LIN {X 0,Y 128.631,Z 703.14,A -85,B 0,C 180,E1 -30051.999,E2 -30051.999} C_VEL
LIN {X 0,Y 134.628,Z 692.341,A -85,B 0,C 180,E1 -30052.672,E2 -30052.672} C_VEL
LIN {X 0,Y 139.361,Z 682.091,A -85,B 0,C 180,E1 -30053.131,E2 -30053.131} C_VEL
LIN {X 0,Y 143.551,Z 670.824,A -85,B 0,C 180,E1 -30053.508,E2 -30053.508} C_VEL
LIN {X 0,Y 146.834,Z 659.297,A -85,B 0,C 180,E1 -30053.808,E2 -30053.808} C_VEL
LIN {X 0,Y 148.842,Z 649.788,A -85,B 0,C 180,E1 -30054.037,E2 -30054.037} C_VEL
LIN {X 0,Y 148.62,Z 648.347,A -85,B 0,C 180,E1 -30055.938,E2 -30055.938} C_VEL
LIN {X 0,Y 148.514,Z 646.401,A -85,B 0,C 180,E1 -30059.999,E2 -30059.999} C_VEL
LIN {X 0,Y 148.714,Z 649.137,A -85,B 0,C 180,E1 -30065.592,E2 -30065.592} C_VEL
LIN {X 0,Y 149.267,Z 652.354,A -85,B 0,C 180,E1 -30069.107,E2 -30069.107} C_VEL
LIN {X 0,Y 149.738,Z 657.139,A -85,B 0,C 180,E1 -30072.527,E2 -30072.527} C_VEL
LIN {X 0,Y 150.095,Z 661.69,A -85,B 0,C 180,E1 -30074.922,E2 -30074.922} C_VEL
LIN {X 0,Y 149.921,Z 667.758,A -85,B 0,C 180,E1 -30077.387,E2 -30077.387} C_VEL
LIN {X 0,Y 149.394,Z 677.527,A -85,B 0,C 180,E1 -30081.047,E2 -30081.047} C_VEL
LIN {X 0,Y 149.068,Z 687.198,A -85,B 0,C 180,E1 -30085.106,E2 -30085.106} C_VEL
LIN {X 0,Y 149.259,Z 696.603,A -85,B 0,C 180,E1 -30089.604,E2 -30089.604} C_VEL
LIN {X 0,Y 150.212,Z 704.997,A -85,B 0,C 180,E1 -30094.154,E2 -30094.154} C_VEL
LIN {X 0,Y 152.27,Z 713.653,A -85,B 0,C 180,E1 -30099.39,E2 -30099.39} C_VEL
LIN {X 0,Y 155.461,Z 721.258,A -85,B 0,C 180,E1 -30104.481,E2 -30104.481} C_VEL
LIN {X 0,Y 160.455,Z 728.846,A -85,B 0,C 180,E1 -30110.039,E2 -30110.039} C_VEL
LIN {X 0,Y 167.763,Z 736.335,A -85,B 0,C 180,E1 -30115.979,E2 -30115.979} C_VEL
LIN {X 0,Y 169.712,Z 738.673,A -85,B 0,C 180,E1 -30117.709,E2 -30117.709} C_VEL
LIN {X 0,Y 173.531,Z 746.392,A -85,B 0,C 180,E1 -30122.934,E2 -30122.934} C_VEL
LIN {X 0,Y 176.298,Z 748.654,A -85,B 0,C 180,E1 -30124.847,E2 -30124.847} C_VEL
LIN {X 0,Y 176.824,Z 748.877,A -85,B 0,C 180,E1 -30125.101,E2 -30125.101} C_VEL
LIN {X 0,Y 192.712,Z 754.942,A -85,B 0,C 180,E1 -30131.472,E2 -30131.472} C_VEL
LIN {X 0,Y 203.581,Z 758.254,A -85,B 0,C 180,E1 -30135.149,E2 -30135.149} C_VEL
LIN {X 0,Y 209.199,Z 759.811,A -85,B 0,C 180,E1 -30136.965,E2 -30136.965} C_VEL
LIN {X 0,Y 214.899,Z 761.328,A -85,B 0,C 180,E1 -30138.841,E2 -30138.841} C_VEL
LIN {X 0,Y 220.679,Z 762.865,A -85,B 0,C 180,E1 -30140.838,E2 -30140.838} C_VEL
LIN {X 0,Y 226.507,Z 764.368,A -85,B 0,C 180,E1 -30143.153,E2 -30143.153} C_VEL
LIN {X 0,Y 229.657,Z 765.23,A -85,B 0,C 180,E1 -30144.733,E2 -30144.733} C_VEL
LIN {X 0,Y 232.744,Z 765.966,A -85,B 0,C 180,E1 -30146.538,E2 -30146.538} C_VEL
LIN {X 0,Y 234.8,Z 766.382,A -85,B 0,C 180,E1 -30148.285,E2 -30148.285} C_VEL
LIN {X 0,Y 236.127,Z 766.522,A -85,B 0,C 180,E1 -30150,E2 -30150} C_VEL
LIN {X 0,Y 234.811,Z 766.381,A -85,B 0,C 180,E1 -30151.715,E2 -30151.715} C_VEL
LIN {X 0,Y 232.396,Z 765.889,A -85,B 0,C 180,E1 -30153.669,E2 -30153.669} C_VEL
LIN {X 0,Y 229.683,Z 765.23,A -85,B 0,C 180,E1 -30155.267,E2 -30155.267} C_VEL
LIN {X 0,Y 225.823,Z 764.189,A -85,B 0,C 180,E1 -30157.151,E2 -30157.151} C_VEL
LIN {X 0,Y 220.686,Z 762.857,A -85,B 0,C 180,E1 -30159.173,E2 -30159.173} C_VEL
LIN {X 0,Y 214.372,Z 761.188,A -85,B 0,C 180,E1 -30161.344,E2 -30161.344} C_VEL
LIN {X 0,Y 207.029,Z 759.205,A -85,B 0,C 180,E1 -30163.746,E2 -30163.746} C_VEL
LIN {X 0,Y 198.092,Z 756.646,A -85,B 0,C 180,E1 -30166.685,E2 -30166.685} C_VEL
LIN {X 0,Y 182.466,Z 751.292,A -85,B 0,C 180,E1 -30172.425,E2 -30172.425} C_VEL
LIN {X 0,Y 170.882,Z 745.936,A -85,B 0,C 180,E1 -30177.844,E2 -30177.844} C_VEL
LIN {X 0,Y 161.108,Z 739.323,A -85,B 0,C 180,E1 -30184.023,E2 -30184.023} C_VEL
LIN {X 0,Y 154.807,Z 733.026,A -85,B 0,C 180,E1 -30189.489,E2 -30189.489} C_VEL
LIN {X 0,Y 149.927,Z 725.802,A -85,B 0,C 180,E1 -30195.322,E2 -30195.322} C_VEL
LIN {X 0,Y 146.606,Z 717.429,A -85,B 0,C 180,E1 -30201.452,E2 -30201.452} C_VEL
LIN {X 0,Y 145.012,Z 708.707,A -85,B 0,C 180,E1 -30207.116,E2 -30207.116} C_VEL
LIN {X 0,Y 144.615,Z 699.602,A -85,B 0,C 180,E1 -30212.333,E2 -30212.333} C_VEL
LIN {X 0,Y 145.085,Z 690.28,A -85,B 0,C 180,E1 -30216.978,E2 -30216.978} C_VEL
LIN {X 0,Y 146.009,Z 680.966,A -85,B 0,C 180,E1 -30221.042,E2 -30221.042} C_VEL
LIN {X 0,Y 147.298,Z 669.426,A -85,B 0,C 180,E1 -30225.494,E2 -30225.494} C_VEL
LIN {X 0,Y 147.568,Z 663.711,A -85,B 0,C 180,E1 -30228.324,E2 -30228.324} C_VEL
LIN {X 0,Y 147.397,Z 659.445,A -85,B 0,C 180,E1 -30231.259,E2 -30231.259} C_VEL
LIN {X 0,Y 147.172,Z 656.298,A -85,B 0,C 180,E1 -30234.521,E2 -30234.521} C_VEL
LIN {X 0,Y 147.108,Z 654.875,A -85,B 0,C 180,E1 -30236.826,E2 -30236.826} C_VEL
LIN {X 0,Y 147.268,Z 653.504,A -85,B 0,C 180,E1 -30240.001,E2 -30240.001} C_VEL
LIN {X 0,Y 147.194,Z 655.069,A -85,B 0,C 180,E1 -30243.318,E2 -30243.318} C_VEL
LIN {X 0,Y 144.031,Z 667.176,A -85,B 0,C 180,E1 -30243.612,E2 -30243.612} C_VEL
LIN {X 0,Y 140,Z 678.676,A -85,B 0,C 180,E1 -30243.883,E2 -30243.883} C_VEL
LIN {X 0,Y 135.652,Z 688.64,A -85,B 0,C 180,E1 -30244.21,E2 -30244.21} C_VEL
LIN {X 0,Y 130.439,Z 698.552,A -85,B 0,C 180,E1 -30244.623,E2 -30244.623} C_VEL
LIN {X 0,Y 124.375,Z 708.269,A -85,B 0,C 180,E1 -30245.188,E2 -30245.188} C_VEL
LIN {X 0,Y 117.455,Z 717.679,A -85,B 0,C 180,E1 -30245.875,E2 -30245.875} C_VEL
LIN {X 0,Y 109.709,Z 726.693,A -85,B 0,C 180,E1 -30246.824,E2 -30246.824} C_VEL
LIN {X 0,Y 102.486,Z 734.008,A -85,B 0,C 180,E1 -30247.885,E2 -30247.885} C_VEL
LIN {X 0,Y 94.355,Z 741.184,A -85,B 0,C 180,E1 -30249.286,E2 -30249.286} C_VEL
LIN {X 0,Y 84.224,Z 748.79,A -85,B 0,C 180,E1 -30251.351,E2 -30251.351} C_VEL
LIN {X 0,Y 75.887,Z 754.19,A -85,B 0,C 180,E1 -30253.495,E2 -30253.495} C_VEL
LIN {X 0,Y 66.094,Z 759.623,A -85,B 0,C 180,E1 -30256.868,E2 -30256.868} C_VEL
LIN {X 0,Y 56.618,Z 764.075,A -85,B 0,C 180,E1 -30261.425,E2 -30261.425} C_VEL
LIN {X 0,Y 47.658,Z 767.628,A -85,B 0,C 180,E1 -30267.776,E2 -30267.776} C_VEL
LIN {X 0,Y 42.078,Z 769.575,A -85,B 0,C 180,E1 -30273.374,E2 -30273.374} C_VEL
LIN {X 0,Y 32.641,Z 772.279,A -85,B 0,C 180,E1 -30289.766,E2 -30289.766} C_VEL
LIN {X 0,Y 27.433,Z 773.598,A -85,B 0,C 180,E1 -30315.156,E2 -30315.156} C_VEL
LIN {X 0,Y 27.054,Z 773.863,A -85,B 0,C 180,E1 -30330,E2 -30330} C_VEL
LIN {X 0,Y 29.383,Z 773.111,A -85,B 0,C 180,E1 -30358.578,E2 -30358.578} C_VEL
LIN {X 0,Y 32.641,Z 772.279,A -85,B 0,C 180,E1 -30370.235,E2 -30370.235} C_VEL
LIN {X 0,Y 42.073,Z 769.575,A -85,B 0,C 180,E1 -30386.635,E2 -30386.635} C_VEL
LIN {X 0,Y 50.55,Z 766.607,A -85,B 0,C 180,E1 -30394.645,E2 -30394.645} C_VEL
LIN {X 0,Y 59.739,Z 762.774,A -85,B 0,C 180,E1 -30400.245,E2 -30400.245} C_VEL
LIN {X 0,Y 69.33,Z 758.007,A -85,B 0,C 180,E1 -30404.364,E2 -30404.364} C_VEL
LIN {X 0,Y 80.868,Z 751.063,A -85,B 0,C 180,E1 -30407.872,E2 -30407.872} C_VEL
LIN {X 0,Y 90.975,Z 743.859,A -85,B 0,C 180,E1 -30410.044,E2 -30410.044} C_VEL
LIN {X 0,Y 99.476,Z 736.792,A -85,B 0,C 180,E1 -30411.523,E2 -30411.523} C_VEL
LIN {X 0,Y 108.005,Z 728.514,A -85,B 0,C 180,E1 -30412.891,E2 -30412.891} C_VEL
LIN {X 0,Y 115.737,Z 719.798,A -85,B 0,C 180,E1 -30413.895,E2 -30413.895} C_VEL
LIN {X 0,Y 122.643,Z 710.747,A -85,B 0,C 180,E1 -30414.652,E2 -30414.652} C_VEL
LIN {X 0,Y 128.704,Z 701.478,A -85,B 0,C 180,E1 -30415.231,E2 -30415.231} C_VEL
LIN {X 0,Y 133.909,Z 692.143,A -85,B 0,C 180,E1 -30415.684,E2 -30415.684} C_VEL
LIN {X 0,Y 138.692,Z 681.893,A -85,B 0,C 180,E1 -30416.039,E2 -30416.039} C_VEL
LIN {X 0,Y 142.851,Z 670.851,A -85,B 0,C 180,E1 -30416.328,E2 -30416.328} C_VEL
LIN {X 0,Y 146.112,Z 659.636,A -85,B 0,C 180,E1 -30416.56,E2 -30416.56} C_VEL
LIN {X 0,Y 147.191,Z 655.075,A -85,B 0,C 180,E1 -30416.691,E2 -30416.691} C_VEL
LIN {X 0,Y 147.269,Z 653.498,A -85,B 0,C 180,E1 -30419.999,E2 -30419.999} C_VEL
LIN {X 0,Y 147.164,Z 655.943,A -85,B 0,C 180,E1 -30425.05,E2 -30425.05} C_VEL
LIN {X 0,Y 147.363,Z 658.957,A -85,B 0,C 180,E1 -30428.326,E2 -30428.326} C_VEL
LIN {X 0,Y 147.578,Z 662.572,A -85,B 0,C 180,E1 -30430.98,E2 -30430.98} C_VEL
LIN {X 0,Y 147.465,Z 666.324,A -85,B 0,C 180,E1 -30433.083,E2 -30433.083} C_VEL
LIN {X 0,Y 147.16,Z 671.262,A -85,B 0,C 180,E1 -30435.228,E2 -30435.228} C_VEL
LIN {X 0,Y 145.677,Z 684.666,A -85,B 0,C 180,E1 -30440.529,E2 -30440.529} C_VEL
LIN {X 0,Y 144.86,Z 694.637,A -85,B 0,C 180,E1 -30445.118,E2 -30445.118} C_VEL
LIN {X 0,Y 144.752,Z 704.962,A -85,B 0,C 180,E1 -30450.649,E2 -30450.649} C_VEL
LIN {X 0,Y 145.787,Z 713.972,A -85,B 0,C 180,E1 -30456.193,E2 -30456.193} C_VEL
LIN {X 0,Y 148.483,Z 722.834,A -85,B 0,C 180,E1 -30462.412,E2 -30462.412} C_VEL
LIN {X 0,Y 152.199,Z 729.57,A -85,B 0,C 180,E1 -30467.629,E2 -30467.629} C_VEL
LIN {X 0,Y 158.771,Z 737.265,A -85,B 0,C 180,E1 -30474.127,E2 -30474.127} C_VEL
LIN {X 0,Y 166.3,Z 743.228,A -85,B 0,C 180,E1 -30479.528,E2 -30479.528} C_VEL
LIN {X 0,Y 176.824,Z 748.877,A -85,B 0,C 180,E1 -30485.101,E2 -30485.101} C_VEL
LIN {X 0,Y 179.618,Z 750.606,A -85,B 0,C 180,E1 -30486.682,E2 -30486.682} C_VEL
LIN {X 0,Y 182.983,Z 753.911,A -85,B 0,C 180,E1 -30489.444,E2 -30489.444} C_VEL
LIN {X 0,Y 185.814,Z 756.293,A -85,B 0,C 180,E1 -30491.622,E2 -30491.622} C_VEL
LIN {X 0,Y 188.736,Z 757.733,A -85,B 0,C 180,E1 -30493.13,E2 -30493.13} C_VEL
LIN {X 0,Y 189.939,Z 758.098,A -85,B 0,C 180,E1 -30493.587,E2 -30493.587} C_VEL
LIN {X 0,Y 203.479,Z 761.495,A -85,B 0,C 180,E1 -30498.04,E2 -30498.04} C_VEL
LIN {X 0,Y 210.566,Z 763.153,A -85,B 0,C 180,E1 -30500.394,E2 -30500.394} C_VEL
LIN {X 0,Y 216.571,Z 764.444,A -85,B 0,C 180,E1 -30502.542,E2 -30502.542} C_VEL
LIN {X 0,Y 219.238,Z 764.993,A -85,B 0,C 180,E1 -30503.582,E2 -30503.582} C_VEL
LIN {X 0,Y 221.312,Z 765.463,A -85,B 0,C 180,E1 -30504.533,E2 -30504.533} C_VEL
LIN {X 0,Y 225.271,Z 766.252,A -85,B 0,C 180,E1 -30506.676,E2 -30506.676} C_VEL
LIN {X 0,Y 227.318,Z 766.587,A -85,B 0,C 180,E1 -30508.228,E2 -30508.228} C_VEL
LIN {X 0,Y 228.896,Z 766.724,A -85,B 0,C 180,E1 -30510,E2 -30510} C_VEL
LIN {X 0,Y 227.327,Z 766.587,A -85,B 0,C 180,E1 -30511.772,E2 -30511.772} C_VEL
LIN {X 0,Y 224.825,Z 766.187,A -85,B 0,C 180,E1 -30513.584,E2 -30513.584} C_VEL
LIN {X 0,Y 221.344,Z 765.462,A -85,B 0,C 180,E1 -30515.466,E2 -30515.466} C_VEL
LIN {X 0,Y 219.24,Z 764.99,A -85,B 0,C 180,E1 -30516.423,E2 -30516.423} C_VEL
LIN {X 0,Y 213.274,Z 763.724,A -85,B 0,C 180,E1 -30518.673,E2 -30518.673} C_VEL
LIN {X 0,Y 207.394,Z 762.392,A -85,B 0,C 180,E1 -30520.671,E2 -30520.671} C_VEL
LIN {X 0,Y 201.614,Z 761.075,A -85,B 0,C 180,E1 -30522.572,E2 -30522.572} C_VEL
LIN {X 0,Y 186.877,Z 757.241,A -85,B 0,C 180,E1 -30527.509,E2 -30527.509} C_VEL
LIN {X 0,Y 169.88,Z 751.256,A -85,B 0,C 180,E1 -30534.477,E2 -30534.477} C_VEL
LIN {X 0,Y 159.155,Z 745.601,A -85,B 0,C 180,E1 -30540.564,E2 -30540.564} C_VEL
LIN {X 0,Y 152.043,Z 740.176,A -85,B 0,C 180,E1 -30546.014,E2 -30546.014} C_VEL
LIN {X 0,Y 146.258,Z 733.384,A -85,B 0,C 180,E1 -30552.277,E2 -30552.277} C_VEL
LIN {X 0,Y 142.626,Z 726.672,A -85,B 0,C 180,E1 -30558.024,E2 -30558.024} C_VEL
LIN {X 0,Y 140.256,Z 717.486,A -85,B 0,C 180,E1 -30564.975,E2 -30564.975} C_VEL
LIN {X 0,Y 139.769,Z 710.287,A -85,B 0,C 180,E1 -30569.814,E2 -30569.814} C_VEL
LIN {X 0,Y 140.326,Z 700.581,A -85,B 0,C 180,E1 -30575.449,E2 -30575.449} C_VEL
LIN {X 0,Y 141.669,Z 690.542,A -85,B 0,C 180,E1 -30580.482,E2 -30580.482} C_VEL
LIN {X 0,Y 143.465,Z 680.267,A -85,B 0,C 180,E1 -30584.866,E2 -30584.866} C_VEL
LIN {X 0,Y 144.643,Z 673.944,A -85,B 0,C 180,E1 -30587.37,E2 -30587.37} C_VEL
LIN {X 0,Y 145.048,Z 669.625,A -85,B 0,C 180,E1 -30589.533,E2 -30589.533} C_VEL
LIN {X 0,Y 145.232,Z 666.495,A -85,B 0,C 180,E1 -30591.654,E2 -30591.654} C_VEL
LIN {X 0,Y 145.396,Z 663.266,A -85,B 0,C 180,E1 -30594.801,E2 -30594.801} C_VEL
LIN {X 0,Y 145.418,Z 661.848,A -85,B 0,C 180,E1 -30596.885,E2 -30596.885} C_VEL
LIN {X 0,Y 145.57,Z 660.548,A -85,B 0,C 180,E1 -30600.001,E2 -30600.001} C_VEL
LIN {X 0,Y 145.51,Z 660.875,A -85,B 0,C 180,E1 -30600.627,E2 -30600.627} C_VEL
LIN {X 0,Y 141.261,Z 674.629,A -85,B 0,C 180,E1 -30600.91,E2 -30600.91} C_VEL
LIN {X 0,Y 136.192,Z 686.69,A -85,B 0,C 180,E1 -30601.165,E2 -30601.165} C_VEL
LIN {X 0,Y 130.06,Z 698.354,A -85,B 0,C 180,E1 -30601.506,E2 -30601.506} C_VEL
LIN {X 0,Y 123.935,Z 708.071,A -85,B 0,C 180,E1 -30601.914,E2 -30601.914} C_VEL
LIN {X 0,Y 116.942,Z 717.481,A -85,B 0,C 180,E1 -30602.418,E2 -30602.418} C_VEL
LIN {X 0,Y 109.091,Z 726.494,A -85,B 0,C 180,E1 -30603.102,E2 -30603.102} C_VEL
LIN {X 0,Y 100.922,Z 734.556,A -85,B 0,C 180,E1 -30603.995,E2 -30603.995} C_VEL
LIN {X 0,Y 93.471,Z 740.986,A -85,B 0,C 180,E1 -30604.975,E2 -30604.975} C_VEL
LIN {X 0,Y 84.837,Z 747.455,A -85,B 0,C 180,E1 -30606.243,E2 -30606.243} C_VEL
LIN {X 0,Y 74.545,Z 753.99,A -85,B 0,C 180,E1 -30608.151,E2 -30608.151} C_VEL
LIN {X 0,Y 64.384,Z 759.424,A -85,B 0,C 180,E1 -30610.769,E2 -30610.769} C_VEL
LIN {X 0,Y 54.417,Z 763.874,A -85,B 0,C 180,E1 -30614.394,E2 -30614.394} C_VEL
LIN {X 0,Y 44.777,Z 767.429,A -85,B 0,C 180,E1 -30619.661,E2 -30619.661} C_VEL
LIN {X 0,Y 38.604,Z 769.376,A -85,B 0,C 180,E1 -30624.462,E2 -30624.462} C_VEL
LIN {X 0,Y 27.568,Z 772.08,A -85,B 0,C 180,E1 -30640.112,E2 -30640.112} C_VEL
LIN {X 0,Y 20.629,Z 773.399,A -85,B 0,C 180,E1 -30670.082,E2 -30670.082} C_VEL
LIN {X 0,Y 19.957,Z 773.665,A -85,B 0,C 180,E1 -30690,E2 -30690} C_VEL
LIN {X 0,Y 23.362,Z 772.912,A -85,B 0,C 180,E1 -30726.987,E2 -30726.987} C_VEL
LIN {X 0,Y 27.567,Z 772.08,A -85,B 0,C 180,E1 -30739.89,E2 -30739.89} C_VEL
LIN {X 0,Y 38.6,Z 769.375,A -85,B 0,C 180,E1 -30755.554,E2 -30755.554} C_VEL
LIN {X 0,Y 51.133,Z 765.141,A -85,B 0,C 180,E1 -30764.174,E2 -30764.174} C_VEL
LIN {X 0,Y 61.036,Z 761.004,A -85,B 0,C 180,E1 -30768.156,E2 -30768.156} C_VEL
LIN {X 0,Y 71.146,Z 755.904,A -85,B 0,C 180,E1 -30771.044,E2 -30771.044} C_VEL
LIN {X 0,Y 81.395,Z 749.728,A -85,B 0,C 180,E1 -30773.185,E2 -30773.185} C_VEL
LIN {X 0,Y 90.014,Z 743.659,A -85,B 0,C 180,E1 -30774.534,E2 -30774.534} C_VEL
LIN {X 0,Y 98.677,Z 736.593,A -85,B 0,C 180,E1 -30775.628,E2 -30775.628} C_VEL
LIN {X 0,Y 107.355,Z 728.314,A -85,B 0,C 180,E1 -30776.676,E2 -30776.676} C_VEL
LIN {X 0,Y 115.198,Z 719.6,A -85,B 0,C 180,E1 -30777.419,E2 -30777.419} C_VEL
LIN {X 0,Y 122.185,Z 710.549,A -85,B 0,C 180,E1 -30777.97,E2 -30777.97} C_VEL
LIN {X 0,Y 128.308,Z 701.28,A -85,B 0,C 180,E1 -30778.396,E2 -30778.396} C_VEL
LIN {X 0,Y 133.562,Z 691.945,A -85,B 0,C 180,E1 -30778.717,E2 -30778.717} C_VEL
LIN {X 0,Y 138.383,Z 681.695,A -85,B 0,C 180,E1 -30778.968,E2 -30778.968} C_VEL
LIN {X 0,Y 142.572,Z 670.653,A -85,B 0,C 180,E1 -30779.178,E2 -30779.178} C_VEL
LIN {X 0,Y 145.516,Z 660.849,A -85,B 0,C 180,E1 -30779.382,E2 -30779.382} C_VEL
LIN {X 0,Y 145.572,Z 660.537,A -85,B 0,C 180,E1 -30779.999,E2 -30779.999} C_VEL
LIN {X 0,Y 145.418,Z 662.581,A -85,B 0,C 180,E1 -30784.329,E2 -30784.329} C_VEL
LIN {X 0,Y 145.32,Z 664.859,A -85,B 0,C 180,E1 -30786.943,E2 -30786.943} C_VEL
LIN {X 0,Y 145.126,Z 668.458,A -85,B 0,C 180,E1 -30789.757,E2 -30789.757} C_VEL
LIN {X 0,Y 144.82,Z 672.393,A -85,B 0,C 180,E1 -30791.902,E2 -30791.902} C_VEL
LIN {X 0,Y 143.686,Z 678.991,A -85,B 0,C 180,E1 -30794.632,E2 -30794.632} C_VEL
LIN {X 0,Y 142.28,Z 687.049,A -85,B 0,C 180,E1 -30797.982,E2 -30797.982} C_VEL
LIN {X 0,Y 140.872,Z 696.007,A -85,B 0,C 180,E1 -30802.148,E2 -30802.148} C_VEL
LIN {X 0,Y 139.975,Z 704.777,A -85,B 0,C 180,E1 -30806.863,E2 -30806.863} C_VEL
LIN {X 0,Y 139.94,Z 713.697,A -85,B 0,C 180,E1 -30812.417,E2 -30812.417} C_VEL
LIN {X 0,Y 141.228,Z 722.184,A -85,B 0,C 180,E1 -30818.462,E2 -30818.462} C_VEL
LIN {X 0,Y 144.302,Z 730.211,A -85,B 0,C 180,E1 -30824.924,E2 -30824.924} C_VEL
LIN {X 0,Y 149.549,Z 737.581,A -85,B 0,C 180,E1 -30831.528,E2 -30831.528} C_VEL
LIN {X 0,Y 157.24,Z 744.344,A -85,B 0,C 180,E1 -30838.125,E2 -30838.125} C_VEL
LIN {X 0,Y 165.348,Z 749.19,A -85,B 0,C 180,E1 -30843.197,E2 -30843.197} C_VEL
LIN {X 0,Y 179.718,Z 754.967,A -85,B 0,C 180,E1 -30849.804,E2 -30849.804} C_VEL
LIN {X 0,Y 189.939,Z 758.098,A -85,B 0,C 180,E1 -30853.587,E2 -30853.587} C_VEL
LIN {X 0,Y 193.227,Z 759.332,A -85,B 0,C 180,E1 -30855.009,E2 -30855.009} C_VEL
LIN {X 0,Y 197.256,Z 761.606,A -85,B 0,C 180,E1 -30857.586,E2 -30857.586} C_VEL
LIN {X 0,Y 200.448,Z 763.225,A -85,B 0,C 180,E1 -30859.649,E2 -30859.649} C_VEL
LIN {X 0,Y 203.53,Z 764.126,A -85,B 0,C 180,E1 -30861.073,E2 -30861.073} C_VEL
LIN {X 0,Y 204.766,Z 764.344,A -85,B 0,C 180,E1 -30861.504,E2 -30861.504} C_VEL
LIN {X 0,Y 212.563,Z 765.707,A -85,B 0,C 180,E1 -30864.308,E2 -30864.308} C_VEL
LIN {X 0,Y 218.151,Z 766.587,A -85,B 0,C 180,E1 -30867.06,E2 -30867.06} C_VEL
LIN {X 0,Y 219.75,Z 766.795,A -85,B 0,C 180,E1 -30868.167,E2 -30868.167} C_VEL
LIN {X 0,Y 221.6,Z 766.928,A -85,B 0,C 180,E1 -30870,E2 -30870} C_VEL
LIN {X 0,Y 219.757,Z 766.795,A -85,B 0,C 180,E1 -30871.833,E2 -30871.833} C_VEL
LIN {X 0,Y 218.152,Z 766.586,A -85,B 0,C 180,E1 -30872.944,E2 -30872.944} C_VEL
LIN {X 0,Y 212.582,Z 765.707,A -85,B 0,C 180,E1 -30875.692,E2 -30875.692} C_VEL
LIN {X 0,Y 205.884,Z 764.541,A -85,B 0,C 180,E1 -30878.143,E2 -30878.143} C_VEL
LIN {X 0,Y 199.893,Z 763.456,A -85,B 0,C 180,E1 -30880.125,E2 -30880.125} C_VEL
LIN {X 0,Y 188.242,Z 761.032,A -85,B 0,C 180,E1 -30883.907,E2 -30883.907} C_VEL
LIN {X 0,Y 171.918,Z 756.706,A -85,B 0,C 180,E1 -30889.912,E2 -30889.912} C_VEL
LIN {X 0,Y 158.651,Z 751.655,A -85,B 0,C 180,E1 -30896.294,E2 -30896.294} C_VEL
LIN {X 0,Y 149.684,Z 746.476,A -85,B 0,C 180,E1 -30902.316,E2 -30902.316} C_VEL
LIN {X 0,Y 143.287,Z 740.908,A -85,B 0,C 180,E1 -30908.303,E2 -30908.303} C_VEL
LIN {X 0,Y 138.151,Z 733.691,A -85,B 0,C 180,E1 -30915.413,E2 -30915.413} C_VEL
LIN {X 0,Y 135.626,Z 726.781,A -85,B 0,C 180,E1 -30921.552,E2 -30921.552} C_VEL
LIN {X 0,Y 134.673,Z 719.516,A -85,B 0,C 180,E1 -30927.311,E2 -30927.311} C_VEL
LIN {X 0,Y 135.021,Z 710.638,A -85,B 0,C 180,E1 -30933.432,E2 -30933.432} C_VEL
LIN {X 0,Y 136.489,Z 701.373,A -85,B 0,C 180,E1 -30938.874,E2 -30938.874} C_VEL
LIN {X 0,Y 138.862,Z 690.799,A -85,B 0,C 180,E1 -30944.069,E2 -30944.069} C_VEL
LIN {X 0,Y 141.45,Z 680.186,A -85,B 0,C 180,E1 -30948.538,E2 -30948.538} C_VEL
LIN {X 0,Y 142.159,Z 676.902,A -85,B 0,C 180,E1 -30950.039,E2 -30950.039} C_VEL
LIN {X 0,Y 142.661,Z 674.363,A -85,B 0,C 180,E1 -30951.502,E2 -30951.502} C_VEL
LIN {X 0,Y 143.055,Z 670.804,A -85,B 0,C 180,E1 -30954.363,E2 -30954.363} C_VEL
LIN {X 0,Y 143.314,Z 668.594,A -85,B 0,C 180,E1 -30957.19,E2 -30957.19} C_VEL
LIN {X 0,Y 143.336,Z 668.409,A -85,B 0,C 180,E1 -30957.606,E2 -30957.606} C_VEL
LIN {X 0,Y 142.719,Z 670.227,A -85,B 0,C 180,E1 -30957.994,E2 -30957.994} C_VEL
LIN {X 0,Y 138.409,Z 681.566,A -85,B 0,C 180,E1 -30958.094,E2 -30958.094} C_VEL
LIN {X 0,Y 131.829,Z 695.202,A -85,B 0,C 180,E1 -30958.309,E2 -30958.309} C_VEL
LIN {X 0,Y 123.902,Z 707.872,A -85,B 0,C 180,E1 -30958.619,E2 -30958.619} C_VEL
LIN {X 0,Y 116.858,Z 717.283,A -85,B 0,C 180,E1 -30958.931,E2 -30958.931} C_VEL
LIN {X 0,Y 108.938,Z 726.295,A -85,B 0,C 180,E1 -30959.351,E2 -30959.351} C_VEL
LIN {X 0,Y 101.944,Z 733.232,A -85,B 0,C 180,E1 -30959.854,E2 -30959.854} C_VEL
LIN {X 0,Y 93.124,Z 740.787,A -85,B 0,C 180,E1 -30960.612,E2 -30960.612} C_VEL
LIN {X 0,Y 84.36,Z 747.256,A -85,B 0,C 180,E1 -30961.435,E2 -30961.435} C_VEL
LIN {X 0,Y 73.871,Z 753.791,A -85,B 0,C 180,E1 -30962.646,E2 -30962.646} C_VEL
LIN {X 0,Y 63.438,Z 759.224,A -85,B 0,C 180,E1 -30964.401,E2 -30964.401} C_VEL
LIN {X 0,Y 53.093,Z 763.674,A -85,B 0,C 180,E1 -30966.9,E2 -30966.9} C_VEL
LIN {X 0,Y 42.9,Z 767.229,A -85,B 0,C 180,E1 -30970.604,E2 -30970.604} C_VEL
LIN {X 0,Y 36.231,Z 769.176,A -85,B 0,C 180,E1 -30974.1,E2 -30974.1} C_VEL
LIN {X 0,Y 23.602,Z 771.88,A -85,B 0,C 180,E1 -30986.708,E2 -30986.708} C_VEL
LIN {X 0,Y 14.152,Z 773.201,A -85,B 0,C 180,E1 -31020.224,E2 -31020.224} C_VEL
LIN {X 0,Y 12.849,Z 773.467,A -85,B 0,C 180,E1 -31050,E2 -31050} C_VEL
LIN {X 0,Y 18.164,Z 772.713,A -85,B 0,C 180,E1 -31100.7,E2 -31100.7} C_VEL
LIN {X 0,Y 23.601,Z 771.88,A -85,B 0,C 180,E1 -31113.295,E2 -31113.295} C_VEL
LIN {X 0,Y 36.227,Z 769.175,A -85,B 0,C 180,E1 -31125.924,E2 -31125.924} C_VEL
LIN {X 0,Y 49.662,Z 764.941,A -85,B 0,C 180,E1 -31132.134,E2 -31132.134} C_VEL
LIN {X 0,Y 59.977,Z 760.805,A -85,B 0,C 180,E1 -31134.867,E2 -31134.867} C_VEL
LIN {X 0,Y 70.388,Z 755.705,A -85,B 0,C 180,E1 -31136.803,E2 -31136.803} C_VEL
LIN {X 0,Y 80.86,Z 749.529,A -85,B 0,C 180,E1 -31138.207,E2 -31138.207} C_VEL
LIN {X 0,Y 89.616,Z 743.46,A -85,B 0,C 180,E1 -31139.094,E2 -31139.094} C_VEL
LIN {X 0,Y 98.39,Z 736.394,A -85,B 0,C 180,E1 -31139.774,E2 -31139.774} C_VEL
LIN {X 0,Y 105.42,Z 729.933,A -85,B 0,C 180,E1 -31140.363,E2 -31140.363} C_VEL
LIN {X 0,Y 114.217,Z 720.46,A -85,B 0,C 180,E1 -31140.916,E2 -31140.916} C_VEL
LIN {X 0,Y 121.26,Z 711.59,A -85,B 0,C 180,E1 -31141.265,E2 -31141.265} C_VEL
LIN {X 0,Y 127.425,Z 702.546,A -85,B 0,C 180,E1 -31141.529,E2 -31141.529} C_VEL
LIN {X 0,Y 133.592,Z 691.748,A -85,B 0,C 180,E1 -31141.757,E2 -31141.757} C_VEL
LIN {X 0,Y 138.412,Z 681.559,A -85,B 0,C 180,E1 -31141.911,E2 -31141.911} C_VEL
LIN {X 0,Y 142.708,Z 670.266,A -85,B 0,C 180,E1 -31142.037,E2 -31142.037} C_VEL
LIN {X 0,Y 143.343,Z 668.385,A -85,B 0,C 180,E1 -31142.394,E2 -31142.394} C_VEL
LIN {X 0,Y 143.194,Z 669.535,A -85,B 0,C 180,E1 -31144.221,E2 -31144.221} C_VEL
LIN {X 0,Y 142.901,Z 672.393,A -85,B 0,C 180,E1 -31147.061,E2 -31147.061} C_VEL
LIN {X 0,Y 142.414,Z 675.629,A -85,B 0,C 180,E1 -31149.264,E2 -31149.264} C_VEL
LIN {X 0,Y 141.458,Z 680.166,A -85,B 0,C 180,E1 -31151.461,E2 -31151.461} C_VEL
LIN {X 0,Y 139.144,Z 689.568,A -85,B 0,C 180,E1 -31155.376,E2 -31155.376} C_VEL
LIN {X 0,Y 137.038,Z 698.636,A -85,B 0,C 180,E1 -31159.705,E2 -31159.705} C_VEL
LIN {X 0,Y 135.46,Z 707.265,A -85,B 0,C 180,E1 -31164.522,E2 -31164.522} C_VEL
LIN {X 0,Y 134.656,Z 715.358,A -85,B 0,C 180,E1 -31169.723,E2 -31169.723} C_VEL
LIN {X 0,Y 134.876,Z 722.535,A -85,B 0,C 180,E1 -31174.97,E2 -31174.97} C_VEL
LIN {X 0,Y 136.821,Z 730.784,A -85,B 0,C 180,E1 -31181.892,E2 -31181.892} C_VEL
LIN {X 0,Y 140.696,Z 737.792,A -85,B 0,C 180,E1 -31188.525,E2 -31188.525} C_VEL
LIN {X 0,Y 146.384,Z 743.886,A -85,B 0,C 180,E1 -31194.822,E2 -31194.822} C_VEL
LIN {X 0,Y 155.485,Z 750.083,A -85,B 0,C 180,E1 -31201.81,E2 -31201.81} C_VEL
LIN {X 0,Y 166.875,Z 755.021,A -85,B 0,C 180,E1 -31207.898,E2 -31207.898} C_VEL
LIN {X 0,Y 177.173,Z 758.264,A -85,B 0,C 180,E1 -31212.175,E2 -31212.175} C_VEL
LIN {X 0,Y 191.882,Z 761.822,A -85,B 0,C 180,E1 -31217.305,E2 -31217.305} C_VEL
LIN {X 0,Y 199.893,Z 763.456,A -85,B 0,C 180,E1 -31219.875,E2 -31219.875} C_VEL
LIN {X 0,Y 204.766,Z 764.344,A -85,B 0,C 180,E1 -31221.504,E2 -31221.504} C_VEL
LIN {X 0,Y 206.995,Z 764.844,A -85,B 0,C 180,E1 -31222.394,E2 -31222.394} C_VEL
LIN {X 0,Y 209.28,Z 765.642,A -85,B 0,C 180,E1 -31223.884,E2 -31223.884} C_VEL
LIN {X 0,Y 210.699,Z 766.283,A -85,B 0,C 180,E1 -31225.46,E2 -31225.46} C_VEL
LIN {X 0,Y 212.925,Z 767.065,A -85,B 0,C 180,E1 -31228.753,E2 -31228.753} C_VEL
LIN {X 0,Y 214.016,Z 767.121,A -85,B 0,C 180,E1 -31229.821,E2 -31229.821} C_VEL
LIN {X 0,Y 214.233,Z 767.133,A -85,B 0,C 180,E1 -31230,E2 -31230} C_VEL
LIN {X 0,Y 212.053,Z 767.007,A -85,B 0,C 180,E1 -31231.899,E2 -31231.899} C_VEL
LIN {X 0,Y 211.039,Z 766.926,A -85,B 0,C 180,E1 -31232.516,E2 -31232.516} C_VEL
LIN {X 0,Y 208.224,Z 766.647,A -85,B 0,C 180,E1 -31233.871,E2 -31233.871} C_VEL
LIN {X 0,Y 203.024,Z 765.974,A -85,B 0,C 180,E1 -31235.961,E2 -31235.961} C_VEL
LIN {X 0,Y 196.31,Z 765.005,A -85,B 0,C 180,E1 -31238.233,E2 -31238.233} C_VEL
LIN {X 0,Y 186.413,Z 763.383,A -85,B 0,C 180,E1 -31241.418,E2 -31241.418} C_VEL
LIN {X 0,Y 171.243,Z 760.221,A -85,B 0,C 180,E1 -31246.695,E2 -31246.695} C_VEL
LIN {X 0,Y 159.072,Z 756.744,A -85,B 0,C 180,E1 -31251.909,E2 -31251.909} C_VEL
LIN {X 0,Y 147.821,Z 751.99,A -85,B 0,C 180,E1 -31258.387,E2 -31258.387} C_VEL
LIN {X 0,Y 140.931,Z 747.67,A -85,B 0,C 180,E1 -31263.882,E2 -31263.882} C_VEL
LIN {X 0,Y 134.807,Z 741.618,A -85,B 0,C 180,E1 -31270.895,E2 -31270.895} C_VEL
LIN {X 0,Y 130.643,Z 733.993,A -85,B 0,C 180,E1 -31278.861,E2 -31278.861} C_VEL
LIN {X 0,Y 129.254,Z 726.854,A -85,B 0,C 180,E1 -31285.435,E2 -31285.435} C_VEL
LIN {X 0,Y 129.583,Z 718.102,A -85,B 0,C 180,E1 -31292.377,E2 -31292.377} C_VEL
LIN {X 0,Y 131.18,Z 709.762,A -85,B 0,C 180,E1 -31297.976,E2 -31297.976} C_VEL
LIN {X 0,Y 133.577,Z 700.9,A -85,B 0,C 180,E1 -31303.047,E2 -31303.047} C_VEL
LIN {X 0,Y 136.62,Z 691.056,A -85,B 0,C 180,E1 -31307.789,E2 -31307.789} C_VEL
LIN {X 0,Y 139.229,Z 682.834,A -85,B 0,C 180,E1 -31311.291,E2 -31311.291} C_VEL
LIN {X 0,Y 139.878,Z 680.136,A -85,B 0,C 180,E1 -31312.785,E2 -31312.785} C_VEL
LIN {X 0,Y 140.498,Z 677.384,A -85,B 0,C 180,E1 -31314.979,E2 -31314.979} C_VEL
LIN {X 0,Y 139.464,Z 679.816,A -85,B 0,C 180,E1 -31315.168,E2 -31315.168} C_VEL
LIN {X 0,Y 134.71,Z 690.132,A -85,B 0,C 180,E1 -31315.214,E2 -31315.214} C_VEL
LIN {X 0,Y 129.58,Z 699.421,A -85,B 0,C 180,E1 -31315.26,E2 -31315.26} C_VEL
LIN {X 0,Y 123.392,Z 708.913,A -85,B 0,C 180,E1 -31315.356,E2 -31315.356} C_VEL
LIN {X 0,Y 117.207,Z 717.084,A -85,B 0,C 180,E1 -31315.452,E2 -31315.452} C_VEL
LIN {X 0,Y 109.253,Z 726.096,A -85,B 0,C 180,E1 -31315.605,E2 -31315.605} C_VEL
LIN {X 0,Y 101.818,Z 733.38,A -85,B 0,C 180,E1 -31315.861,E2 -31315.861} C_VEL
LIN {X 0,Y 93.319,Z 740.589,A -85,B 0,C 180,E1 -31316.244,E2 -31316.244} C_VEL
LIN {X 0,Y 84.483,Z 747.058,A -85,B 0,C 180,E1 -31316.596,E2 -31316.596} C_VEL
LIN {X 0,Y 73.887,Z 753.591,A -85,B 0,C 180,E1 -31317.103,E2 -31317.103} C_VEL
LIN {X 0,Y 63.291,Z 759.025,A -85,B 0,C 180,E1 -31317.941,E2 -31317.941} C_VEL
LIN {X 0,Y 52.714,Z 763.475,A -85,B 0,C 180,E1 -31319.168,E2 -31319.168} C_VEL
LIN {X 0,Y 42.173,Z 767.029,A -85,B 0,C 180,E1 -31320.998,E2 -31320.998} C_VEL
LIN {X 0,Y 35.179,Z 768.976,A -85,B 0,C 180,E1 -31322.713,E2 -31322.713} C_VEL
LIN {X 0,Y 21.365,Z 771.681,A -85,B 0,C 180,E1 -31329.311,E2 -31329.311} C_VEL
LIN {X 0,Y 8.71,Z 773.002,A -85,B 0,C 180,E1 -31356.205,E2 -31356.205} C_VEL
LIN {X 0,Y 5.734,Z 773.268,A -85,B 0,C 180,E1 -31410,E2 -31410} C_VEL
LIN {X 0,Y 14.715,Z 772.513,A -85,B 0,C 180,E1 -31482.781,E2 -31482.781} C_VEL
LIN {X 0,Y 21.365,Z 771.681,A -85,B 0,C 180,E1 -31490.694,E2 -31490.694} C_VEL
LIN {X 0,Y 35.178,Z 768.976,A -85,B 0,C 180,E1 -31497.318,E2 -31497.318} C_VEL
LIN {X 0,Y 49.196,Z 764.742,A -85,B 0,C 180,E1 -31500.39,E2 -31500.39} C_VEL
LIN {X 0,Y 59.763,Z 760.605,A -85,B 0,C 180,E1 -31501.706,E2 -31501.706} C_VEL
LIN {X 0,Y 70.353,Z 755.505,A -85,B 0,C 180,E1 -31502.642,E2 -31502.642} C_VEL
LIN {X 0,Y 80.951,Z 749.33,A -85,B 0,C 180,E1 -31503.265,E2 -31503.265} C_VEL
LIN {X 0,Y 89.787,Z 743.261,A -85,B 0,C 180,E1 -31503.654,E2 -31503.654} C_VEL
LIN {X 0,Y 98.62,Z 736.195,A -85,B 0,C 180,E1 -31503.913,E2 -31503.913} C_VEL
LIN {X 0,Y 105.706,Z 729.734,A -85,B 0,C 180,E1 -31504.236,E2 -31504.236} C_VEL
LIN {X 0,Y 114.55,Z 720.262,A -85,B 0,C 180,E1 -31504.467,E2 -31504.467} C_VEL
LIN {X 0,Y 121.625,Z 711.392,A -85,B 0,C 180,E1 -31504.618,E2 -31504.618} C_VEL
LIN {X 0,Y 127.813,Z 702.347,A -85,B 0,C 180,E1 -31504.723,E2 -31504.723} C_VEL
LIN {X 0,Y 133.996,Z 691.55,A -85,B 0,C 180,E1 -31504.785,E2 -31504.785} C_VEL
LIN {X 0,Y 138.735,Z 681.595,A -85,B 0,C 180,E1 -31504.844,E2 -31504.844} C_VEL
LIN {X 0,Y 139.893,Z 678.764,A -85,B 0,C 180,E1 -31504.818,E2 -31504.818} C_VEL
LIN {X 0,Y 140.44,Z 677.638,A -85,B 0,C 180,E1 -31505.264,E2 -31505.264} C_VEL
LIN {X 0,Y 139.819,Z 680.39,A -85,B 0,C 180,E1 -31507.377,E2 -31507.377} C_VEL
LIN {X 0,Y 139.231,Z 682.83,A -85,B 0,C 180,E1 -31508.708,E2 -31508.708} C_VEL
LIN {X 0,Y 135.288,Z 695.514,A -85,B 0,C 180,E1 -31514.283,E2 -31514.283} C_VEL
LIN {X 0,Y 132.369,Z 705.317,A -85,B 0,C 180,E1 -31519.379,E2 -31519.379} C_VEL
LIN {X 0,Y 130.043,Z 715.265,A -85,B 0,C 180,E1 -31525.615,E2 -31525.615} C_VEL
LIN {X 0,Y 129.194,Z 723.803,A -85,B 0,C 180,E1 -31532.029,E2 -31532.029} C_VEL
LIN {X 0,Y 129.896,Z 731.211,A -85,B 0,C 180,E1 -31538.475,E2 -31538.475} C_VEL
LIN {X 0,Y 132.565,Z 738.216,A -85,B 0,C 180,E1 -31545.439,E2 -31545.439} C_VEL
LIN {X 0,Y 137.056,Z 744.204,A -85,B 0,C 180,E1 -31552.024,E2 -31552.024} C_VEL
LIN {X 0,Y 143.912,Z 749.774,A -85,B 0,C 180,E1 -31558.715,E2 -31558.715} C_VEL
LIN {X 0,Y 154.311,Z 755.007,A -85,B 0,C 180,E1 -31565.625,E2 -31565.625} C_VEL
LIN {X 0,Y 164.115,Z 758.355,A -85,B 0,C 180,E1 -31570.406,E2 -31570.406} C_VEL
LIN {X 0,Y 180.563,Z 762.283,A -85,B 0,C 180,E1 -31576.667,E2 -31576.667} C_VEL
LIN {X 0,Y 192.385,Z 764.413,A -85,B 0,C 180,E1 -31580.51,E2 -31580.51} C_VEL
LIN {X 0,Y 199.17,Z 765.435,A -85,B 0,C 180,E1 -31582.732,E2 -31582.732} C_VEL
LIN {X 0,Y 204.694,Z 766.173,A -85,B 0,C 180,E1 -31584.667,E2 -31584.667} C_VEL
LIN {X 0,Y 208.207,Z 766.647,A -85,B 0,C 180,E1 -31586.129,E2 -31586.129} C_VEL
LIN {X 0,Y 212.046,Z 767.007,A -85,B 0,C 180,E1 -31588.101,E2 -31588.101} C_VEL
LIN {X 0,Y 214.016,Z 767.121,A -85,B 0,C 180,E1 -31589.821,E2 -31589.821} C_VEL
LIN {X 0,Y 214.115,Z 767.153,A -85,B 0,C 180,E1 -31590.65,E2 -31590.65} C_VEL
LIN {X 0,Y 212.528,Z 767.144,A -85,B 0,C 180,E1 -31591.665,E2 -31591.665} C_VEL
LIN {X 0,Y 208.645,Z 767.06,A -85,B 0,C 180,E1 -31592.869,E2 -31592.869} C_VEL
LIN {X 0,Y 193.952,Z 766.361,A -85,B 0,C 180,E1 -31595.95,E2 -31595.95} C_VEL
LIN {X 0,Y 192.33,Z 766.207,A -85,B 0,C 180,E1 -31596.439,E2 -31596.439} C_VEL
LIN {X 0,Y 184.901,Z 765.288,A -85,B 0,C 180,E1 -31598.8,E2 -31598.8} C_VEL
LIN {X 0,Y 172.905,Z 763.461,A -85,B 0,C 180,E1 -31602.71,E2 -31602.71} C_VEL
LIN {X 0,Y 156.302,Z 759.859,A -85,B 0,C 180,E1 -31609.227,E2 -31609.227} C_VEL
LIN {X 0,Y 143.577,Z 755.52,A -85,B 0,C 180,E1 -31616.138,E2 -31616.138} C_VEL
LIN {X 0,Y 134.56,Z 750.511,A -85,B 0,C 180,E1 -31623.317,E2 -31623.317} C_VEL
LIN {X 0,Y 127.564,Z 743.614,A -85,B 0,C 180,E1 -31632.27,E2 -31632.27} C_VEL
LIN {X 0,Y 124.07,Z 735.421,A -85,B 0,C 180,E1 -31641.459,E2 -31641.459} C_VEL
LIN {X 0,Y 123.658,Z 727.321,A -85,B 0,C 180,E1 -31649.238,E2 -31649.238} C_VEL
LIN {X 0,Y 125.009,Z 719.445,A -85,B 0,C 180,E1 -31655.655,E2 -31655.655} C_VEL
LIN {X 0,Y 127.751,Z 710.371,A -85,B 0,C 180,E1 -31661.798,E2 -31661.798} C_VEL
LIN {X 0,Y 131.045,Z 701.479,A -85,B 0,C 180,E1 -31666.786,E2 -31666.786} C_VEL
LIN {X 0,Y 135,Z 691.308,A -85,B 0,C 180,E1 -31671.535,E2 -31671.535} C_VEL
LIN {X 0,Y 134.775,Z 691.352,A -85,B 0,C 180,E1 -31672.202,E2 -31672.202} C_VEL
LIN {X 0,Y 127.709,Z 703.612,A -85,B 0,C 180,E1 -31672.114,E2 -31672.114} C_VEL
LIN {X 0,Y 118.873,Z 715.826,A -85,B 0,C 180,E1 -31672.001,E2 -31672.001} C_VEL
LIN {X 0,Y 111.797,Z 724.081,A -85,B 0,C 180,E1 -31671.925,E2 -31671.925} C_VEL
LIN {X 0,Y 102.935,Z 732.869,A -85,B 0,C 180,E1 -31671.883,E2 -31671.883} C_VEL
LIN {X 0,Y 93.872,Z 740.528,A -85,B 0,C 180,E1 -31671.916,E2 -31671.916} C_VEL
LIN {X 0,Y 83.436,Z 747.995,A -85,B 0,C 180,E1 -31671.769,E2 -31671.769} C_VEL
LIN {X 0,Y 74.588,Z 753.393,A -85,B 0,C 180,E1 -31671.624,E2 -31671.624} C_VEL
LIN {X 0,Y 63.946,Z 758.826,A -85,B 0,C 180,E1 -31671.541,E2 -31671.541} C_VEL
LIN {X 0,Y 53.301,Z 763.276,A -85,B 0,C 180,E1 -31671.45,E2 -31671.45} C_VEL
LIN {X 0,Y 42.656,Z 766.829,A -85,B 0,C 180,E1 -31671.316,E2 -31671.316} C_VEL
LIN {X 0,Y 35.566,Z 768.777,A -85,B 0,C 180,E1 -31671.119,E2 -31671.119} C_VEL
LIN {X 0,Y 21.405,Z 771.481,A -85,B 0,C 180,E1 -31670.059,E2 -31670.059} C_VEL
LIN {X 0,Y 7.302,Z 772.803,A -85,B 0,C 180,E1 -31664.244,E2 -31664.244} C_VEL
LIN {X 0,Y 1.369,Z 773.07,A -85,B 0,C 180,E1 -31590,E2 -31590} C_VEL
LIN {X 0,Y 14.329,Z 772.314,A -85,B 0,C 180,E1 -31511.199,E2 -31511.199} C_VEL
LIN {X 0,Y 21.405,Z 771.481,A -85,B 0,C 180,E1 -31509.946,E2 -31509.946} C_VEL
LIN {X 0,Y 35.569,Z 768.776,A -85,B 0,C 180,E1 -31508.918,E2 -31508.918} C_VEL
LIN {X 0,Y 45.934,Z 765.902,A -85,B 0,C 180,E1 -31508.797,E2 -31508.797} C_VEL
LIN {X 0,Y 56.851,Z 761.975,A -85,B 0,C 180,E1 -31508.529,E2 -31508.529} C_VEL
LIN {X 0,Y 67.494,Z 757.21,A -85,B 0,C 180,E1 -31508.433,E2 -31508.433} C_VEL
LIN {X 0,Y 79.897,Z 750.268,A -85,B 0,C 180,E1 -31508.285,E2 -31508.285} C_VEL
LIN {X 0,Y 88.747,Z 744.399,A -85,B 0,C 180,E1 -31508.161,E2 -31508.161} C_VEL
LIN {X 0,Y 97.588,Z 737.557,A -85,B 0,C 180,E1 -31508.025,E2 -31508.025} C_VEL
LIN {X 0,Y 106.471,Z 729.535,A -85,B 0,C 180,E1 -31508.068,E2 -31508.068} C_VEL
LIN {X 0,Y 115.324,Z 720.063,A -85,B 0,C 180,E1 -31507.996,E2 -31507.996} C_VEL
LIN {X 0,Y 122.401,Z 711.194,A -85,B 0,C 180,E1 -31507.932,E2 -31507.932} C_VEL
LIN {X 0,Y 128.596,Z 702.148,A -85,B 0,C 180,E1 -31507.886,E2 -31507.886} C_VEL
LIN {X 0,Y 134.772,Z 691.353,A -85,B 0,C 180,E1 -31507.787,E2 -31507.787} C_VEL
LIN {X 0,Y 135,Z 691.308,A -85,B 0,C 180,E1 -31508.468,E2 -31508.468} C_VEL
LIN {X 0,Y 130.441,Z 703.213,A -85,B 0,C 180,E1 -31514.119,E2 -31514.119} C_VEL
LIN {X 0,Y 126.28,Z 714.997,A -85,B 0,C 180,E1 -31521.204,E2 -31521.204} C_VEL
LIN {X 0,Y 124.34,Z 722.728,A -85,B 0,C 180,E1 -31526.882,E2 -31526.882} C_VEL
LIN {X 0,Y 123.569,Z 731.548,A -85,B 0,C 180,E1 -31534.661,E2 -31534.661} C_VEL
LIN {X 0,Y 125.062,Z 738.997,A -85,B 0,C 180,E1 -31542.402,E2 -31542.402} C_VEL
LIN {X 0,Y 128.822,Z 745.226,A -85,B 0,C 180,E1 -31549.796,E2 -31549.796} C_VEL
LIN {X 0,Y 134.57,Z 750.501,A -85,B 0,C 180,E1 -31556.676,E2 -31556.676} C_VEL
LIN {X 0,Y 143.53,Z 755.522,A -85,B 0,C 180,E1 -31563.853,E2 -31563.853} C_VEL
LIN {X 0,Y 156.303,Z 759.858,A -85,B 0,C 180,E1 -31570.772,E2 -31570.772} C_VEL
LIN {X 0,Y 172.897,Z 763.47,A -85,B 0,C 180,E1 -31577.302,E2 -31577.302} C_VEL
LIN {X 0,Y 185.056,Z 765.317,A -85,B 0,C 180,E1 -31581.263,E2 -31581.263} C_VEL
LIN {X 0,Y 192.816,Z 766.259,A -85,B 0,C 180,E1 -31583.722,E2 -31583.722} C_VEL
LIN {X 0,Y 199.222,Z 766.895,A -85,B 0,C 180,E1 -31585.954,E2 -31585.954} C_VEL
LIN {X 0,Y 203.969,Z 767.229,A -85,B 0,C 180,E1 -31588.025,E2 -31588.025} C_VEL
LIN {X 0,Y 206.767,Z 767.341,A -85,B 0,C 180,E1 -31590,E2 -31590} C_VEL
LIN {X 0,Y 203.932,Z 767.226,A -85,B 0,C 180,E1 -31592,E2 -31592} C_VEL
LIN {X 0,Y 199.249,Z 766.895,A -85,B 0,C 180,E1 -31594.045,E2 -31594.045} C_VEL
LIN {X 0,Y 192.33,Z 766.207,A -85,B 0,C 180,E1 -31596.439,E2 -31596.439} C_VEL
LIN {X 0,Y 187.865,Z 765.87,A -85,B 0,C 180,E1 -31597.593,E2 -31597.593} C_VEL
LIN {X 0,Y 182.733,Z 765.648,A -85,B 0,C 180,E1 -31598.519,E2 -31598.519} C_VEL
LIN {X 0,Y 171.986,Z 765.215,A -85,B 0,C 180,E1 -31600.26,E2 -31600.26} C_VEL
LIN {X 0,Y 167.082,Z 764.844,A -85,B 0,C 180,E1 -31601.413,E2 -31601.413} C_VEL
LIN {X 0,Y 165.632,Z 764.657,A -85,B 0,C 180,E1 -31601.881,E2 -31601.881} C_VEL
LIN {X 0,Y 148.5,Z 761.32,A -85,B 0,C 180,E1 -31608.826,E2 -31608.826} C_VEL
LIN {X 0,Y 138.717,Z 758.386,A -85,B 0,C 180,E1 -31614.227,E2 -31614.227} C_VEL
LIN {X 0,Y 130.481,Z 754.625,A -85,B 0,C 180,E1 -31620.485,E2 -31620.485} C_VEL
LIN {X 0,Y 123.148,Z 749.052,A -85,B 0,C 180,E1 -31628.884,E2 -31628.884} C_VEL
LIN {X 0,Y 119.066,Z 742.813,A -85,B 0,C 180,E1 -31637.253,E2 -31637.253} C_VEL
LIN {X 0,Y 117.699,Z 735.808,A -85,B 0,C 180,E1 -31645.445,E2 -31645.445} C_VEL
LIN {X 0,Y 118.788,Z 727.429,A -85,B 0,C 180,E1 -31653.641,E2 -31653.641} C_VEL
LIN {X 0,Y 121.159,Z 720.076,A -85,B 0,C 180,E1 -31659.634,E2 -31659.634} C_VEL
LIN {X 0,Y 125.073,Z 710.723,A -85,B 0,C 180,E1 -31665.88,E2 -31665.88} C_VEL
LIN {X 0,Y 126.95,Z 706.668,A -85,B 0,C 180,E1 -31668.196,E2 -31668.196} C_VEL
LIN {X 0,Y 125.35,Z 708.516,A -85,B 0,C 180,E1 -31668.858,E2 -31668.858} C_VEL
LIN {X 0,Y 119.19,Z 716.686,A -85,B 0,C 180,E1 -31668.598,E2 -31668.598} C_VEL
LIN {X 0,Y 111.255,Z 725.699,A -85,B 0,C 180,E1 -31668.269,E2 -31668.269} C_VEL
LIN {X 0,Y 104.178,Z 732.67,A -85,B 0,C 180,E1 -31668.004,E2 -31668.004} C_VEL
LIN {X 0,Y 94.92,Z 740.491,A -85,B 0,C 180,E1 -31667.66,E2 -31667.66} C_VEL
LIN {X 0,Y 84.75,Z 747.796,A -85,B 0,C 180,E1 -31666.998,E2 -31666.998} C_VEL
LIN {X 0,Y 75.96,Z 753.193,A -85,B 0,C 180,E1 -31666.28,E2 -31666.28} C_VEL
LIN {X 0,Y 65.381,Z 758.627,A -85,B 0,C 180,E1 -31665.333,E2 -31665.333} C_VEL
LIN {X 0,Y 54.826,Z 763.076,A -85,B 0,C 180,E1 -31664.027,E2 -31664.027} C_VEL
LIN {X 0,Y 44.309,Z 766.629,A -85,B 0,C 180,E1 -31662.111,E2 -31662.111} C_VEL
LIN {X 0,Y 37.345,Z 768.577,A -85,B 0,C 180,E1 -31660.209,E2 -31660.209} C_VEL
LIN {X 0,Y 23.71,Z 771.282,A -85,B 0,C 180,E1 -31652.776,E2 -31652.776} C_VEL
LIN {X 0,Y 11.498,Z 772.605,A -85,B 0,C 180,E1 -31627.676,E2 -31627.676} C_VEL
LIN {X 0,Y 8.489,Z 772.872,A -85,B 0,C 180,E1 -31590,E2 -31590} C_VEL
LIN {X 0,Y 17.201,Z 772.115,A -85,B 0,C 180,E1 -31535.198,E2 -31535.198} C_VEL
LIN {X 0,Y 23.711,Z 771.282,A -85,B 0,C 180,E1 -31527.23,E2 -31527.23} C_VEL
LIN {X 0,Y 37.354,Z 768.576,A -85,B 0,C 180,E1 -31519.831,E2 -31519.831} C_VEL
LIN {X 0,Y 46.671,Z 765.976,A -85,B 0,C 180,E1 -31517.524,E2 -31517.524} C_VEL
LIN {X 0,Y 58.344,Z 761.776,A -85,B 0,C 180,E1 -31515.496,E2 -31515.496} C_VEL
LIN {X 0,Y 68.907,Z 757.01,A -85,B 0,C 180,E1 -31514.327,E2 -31514.327} C_VEL
LIN {X 0,Y 81.231,Z 750.07,A -85,B 0,C 180,E1 -31513.265,E2 -31513.265} C_VEL
LIN {X 0,Y 90.041,Z 744.2,A -85,B 0,C 180,E1 -31512.672,E2 -31512.672} C_VEL
LIN {X 0,Y 99.238,Z 737.005,A -85,B 0,C 180,E1 -31512.109,E2 -31512.109} C_VEL
LIN {X 0,Y 107.704,Z 729.336,A -85,B 0,C 180,E1 -31511.827,E2 -31511.827} C_VEL
LIN {X 0,Y 116.527,Z 719.865,A -85,B 0,C 180,E1 -31511.465,E2 -31511.465} C_VEL
LIN {X 0,Y 123.835,Z 710.638,A -85,B 0,C 180,E1 -31511.184,E2 -31511.184} C_VEL
LIN {X 0,Y 125.352,Z 708.516,A -85,B 0,C 180,E1 -31511.146,E2 -31511.146} C_VEL
LIN {X 0,Y 126.987,Z 706.61,A -85,B 0,C 180,E1 -31511.792,E2 -31511.792} C_VEL
LIN {X 0,Y 122.807,Z 715.958,A -85,B 0,C 180,E1 -31517.483,E2 -31517.483} C_VEL
LIN {X 0,Y 119.828,Z 723.864,A -85,B 0,C 180,E1 -31523.319,E2 -31523.319} C_VEL
LIN {X 0,Y 117.962,Z 731.771,A -85,B 0,C 180,E1 -31530.424,E2 -31530.424} C_VEL
LIN {X 0,Y 117.932,Z 738.854,A -85,B 0,C 180,E1 -31537.975,E2 -31537.975} C_VEL
LIN {X 0,Y 120.012,Z 744.823,A -85,B 0,C 180,E1 -31545.355,E2 -31545.355} C_VEL
LIN {X 0,Y 125.49,Z 751.165,A -85,B 0,C 180,E1 -31554.295,E2 -31554.295} C_VEL
LIN {X 0,Y 132.845,Z 755.851,A -85,B 0,C 180,E1 -31561.568,E2 -31561.568} C_VEL
LIN {X 0,Y 143.435,Z 759.919,A -85,B 0,C 180,E1 -31568.58,E2 -31568.58} C_VEL
LIN {X 0,Y 159.435,Z 763.61,A -85,B 0,C 180,E1 -31575.872,E2 -31575.872} C_VEL
LIN {X 0,Y 173.183,Z 765.647,A -85,B 0,C 180,E1 -31580.658,E2 -31580.658} C_VEL
LIN {X 0,Y 183.746,Z 766.719,A -85,B 0,C 180,E1 -31583.955,E2 -31583.955} C_VEL
LIN {X 0,Y 190.209,Z 767.23,A -85,B 0,C 180,E1 -31586.027,E2 -31586.027} C_VEL
LIN {X 0,Y 196.837,Z 767.511,A -85,B 0,C 180,E1 -31588.625,E2 -31588.625} C_VEL
LIN {X 0,Y 199.114,Z 767.555,A -85,B 0,C 180,E1 -31590,E2 -31590} C_VEL
LIN {X 0,Y 196.837,Z 767.509,A -85,B 0,C 180,E1 -31591.387,E2 -31591.387} C_VEL
LIN {X 0,Y 190.21,Z 767.229,A -85,B 0,C 180,E1 -31593.978,E2 -31593.978} C_VEL
LIN {X 0,Y 181.781,Z 766.568,A -85,B 0,C 180,E1 -31596.66,E2 -31596.66} C_VEL
LIN {X 0,Y 171.258,Z 765.406,A -85,B 0,C 180,E1 -31599.978,E2 -31599.978} C_VEL
LIN {X 0,Y 165.632,Z 764.657,A -85,B 0,C 180,E1 -31601.881,E2 -31601.881} C_VEL
LIN {X 0,Y 161.109,Z 764.234,A -85,B 0,C 180,E1 -31603.202,E2 -31603.202} C_VEL
LIN {X 0,Y 152.582,Z 763.84,A -85,B 0,C 180,E1 -31605.045,E2 -31605.045} C_VEL
LIN {X 0,Y 145.785,Z 763.415,A -85,B 0,C 180,E1 -31606.62,E2 -31606.62} C_VEL
LIN {X 0,Y 141.289,Z 762.805,A -85,B 0,C 180,E1 -31608.132,E2 -31608.132} C_VEL
LIN {X 0,Y 140.007,Z 762.518,A -85,B 0,C 180,E1 -31608.73,E2 -31608.73} C_VEL
LIN {X 0,Y 126.612,Z 758.224,A -85,B 0,C 180,E1 -31617.364,E2 -31617.364} C_VEL
LIN {X 0,Y 117.94,Z 752.962,A -85,B 0,C 180,E1 -31626.576,E2 -31626.576} C_VEL
LIN {X 0,Y 113.605,Z 747.839,A -85,B 0,C 180,E1 -31634.651,E2 -31634.651} C_VEL
LIN {X 0,Y 111.737,Z 741.56,A -85,B 0,C 180,E1 -31643.312,E2 -31643.312} C_VEL
LIN {X 0,Y 112.109,Z 736.05,A -85,B 0,C 180,E1 -31649.902,E2 -31649.902} C_VEL
LIN {X 0,Y 114.3,Z 728.72,A -85,B 0,C 180,E1 -31657.263,E2 -31657.263} C_VEL
LIN {X 0,Y 118.472,Z 719.635,A -85,B 0,C 180,E1 -31664.565,E2 -31664.565} C_VEL
LIN {X 0,Y 117.29,Z 720.725,A -85,B 0,C 180,E1 -31665.055,E2 -31665.055} C_VEL
LIN {X 0,Y 107.65,Z 730.901,A -85,B 0,C 180,E1 -31664.354,E2 -31664.354} C_VEL
LIN {X 0,Y 97.321,Z 739.813,A -85,B 0,C 180,E1 -31663.588,E2 -31663.588} C_VEL
LIN {X 0,Y 88.379,Z 746.46,A -85,B 0,C 180,E1 -31662.599,E2 -31662.599} C_VEL
LIN {X 0,Y 77.962,Z 752.994,A -85,B 0,C 180,E1 -31661.176,E2 -31661.176} C_VEL
LIN {X 0,Y 67.552,Z 758.427,A -85,B 0,C 180,E1 -31659.444,E2 -31659.444} C_VEL
LIN {X 0,Y 57.21,Z 762.876,A -85,B 0,C 180,E1 -31657.12,E2 -31657.12} C_VEL
LIN {X 0,Y 47.005,Z 766.429,A -85,B 0,C 180,E1 -31653.776,E2 -31653.776} C_VEL
LIN {X 0,Y 40.331,Z 768.378,A -85,B 0,C 180,E1 -31650.606,E2 -31650.606} C_VEL
LIN {X 0,Y 27.716,Z 771.083,A -85,B 0,C 180,E1 -31639.525,E2 -31639.525} C_VEL
LIN {X 0,Y 17.696,Z 772.406,A -85,B 0,C 180,E1 -31613.399,E2 -31613.399} C_VEL
LIN {X 0,Y 15.596,Z 772.673,A -85,B 0,C 180,E1 -31590,E2 -31590} C_VEL
LIN {X 0,Y 22.105,Z 771.916,A -85,B 0,C 180,E1 -31550.516,E2 -31550.516} C_VEL
LIN {X 0,Y 27.718,Z 771.082,A -85,B 0,C 180,E1 -31540.48,E2 -31540.48} C_VEL
LIN {X 0,Y 40.348,Z 768.377,A -85,B 0,C 180,E1 -31529.436,E2 -31529.436} C_VEL
LIN {X 0,Y 48.401,Z 766.037,A -85,B 0,C 180,E1 -31525.82,E2 -31525.82} C_VEL
LIN {X 0,Y 60.65,Z 761.576,A -85,B 0,C 180,E1 -31522.027,E2 -31522.027} C_VEL
LIN {X 0,Y 71.013,Z 756.811,A -85,B 0,C 180,E1 -31519.92,E2 -31519.92} C_VEL
LIN {X 0,Y 83.163,Z 749.87,A -85,B 0,C 180,E1 -31518.066,E2 -31518.066} C_VEL
LIN {X 0,Y 93.602,Z 742.666,A -85,B 0,C 180,E1 -31516.804,E2 -31516.804} C_VEL
LIN {X 0,Y 102.344,Z 735.597,A -85,B 0,C 180,E1 -31515.979,E2 -31515.979} C_VEL
LIN {X 0,Y 109.39,Z 729.137,A -85,B 0,C 180,E1 -31515.488,E2 -31515.488} C_VEL
LIN {X 0,Y 117.297,Z 720.698,A -85,B 0,C 180,E1 -31514.914,E2 -31514.914} C_VEL
LIN {X 0,Y 118.513,Z 719.579,A -85,B 0,C 180,E1 -31515.421,E2 -31515.421} C_VEL
LIN {X 0,Y 114.3,Z 728.72,A -85,B 0,C 180,E1 -31522.737,E2 -31522.737} C_VEL
LIN {X 0,Y 111.801,Z 738.044,A -85,B 0,C 180,E1 -31532.296,E2 -31532.296} C_VEL
LIN {X 0,Y 112.393,Z 745.126,A -85,B 0,C 180,E1 -31541.379,E2 -31541.379} C_VEL
LIN {X 0,Y 115.512,Z 750.592,A -85,B 0,C 180,E1 -31549.505,E2 -31549.505} C_VEL
LIN {X 0,Y 122.782,Z 756.297,A -85,B 0,C 180,E1 -31559.156,E2 -31559.156} C_VEL
LIN {X 0,Y 130.905,Z 759.903,A -85,B 0,C 180,E1 -31565.876,E2 -31565.876} C_VEL
LIN {X 0,Y 143.215,Z 763.211,A -85,B 0,C 180,E1 -31572.877,E2 -31572.877} C_VEL
LIN {X 0,Y 157.622,Z 765.602,A -85,B 0,C 180,E1 -31578.785,E2 -31578.785} C_VEL
LIN {X 0,Y 169.981,Z 766.897,A -85,B 0,C 180,E1 -31582.875,E2 -31582.875} C_VEL
LIN {X 0,Y 178.626,Z 767.464,A -85,B 0,C 180,E1 -31585.487,E2 -31585.487} C_VEL
LIN {X 0,Y 185.88,Z 767.726,A -85,B 0,C 180,E1 -31587.833,E2 -31587.833} C_VEL
LIN {X 0,Y 189.766,Z 767.766,A -85,B 0,C 180,E1 -31589.291,E2 -31589.291} C_VEL
LIN {X 0,Y 191.214,Z 767.775,A -85,B 0,C 180,E1 -31590,E2 -31590} C_VEL
LIN {X 0,Y 189.767,Z 767.765,A -85,B 0,C 180,E1 -31590.719,E2 -31590.719} C_VEL
LIN {X 0,Y 185.895,Z 767.725,A -85,B 0,C 180,E1 -31592.167,E2 -31592.167} C_VEL
LIN {X 0,Y 178.606,Z 767.465,A -85,B 0,C 180,E1 -31594.514,E2 -31594.514} C_VEL
LIN {X 0,Y 169.986,Z 766.893,A -85,B 0,C 180,E1 -31597.138,E2 -31597.138} C_VEL
LIN {X 0,Y 151.739,Z 764.796,A -85,B 0,C 180,E1 -31603.44,E2 -31603.44} C_VEL
LIN {X 0,Y 140.007,Z 762.518,A -85,B 0,C 180,E1 -31608.73,E2 -31608.73} C_VEL
LIN {X 0,Y 135.962,Z 761.811,A -85,B 0,C 180,E1 -31610.496,E2 -31610.496} C_VEL
LIN {X 0,Y 122.345,Z 760.544,A -85,B 0,C 180,E1 -31615.596,E2 -31615.596} C_VEL
LIN {X 0,Y 118.68,Z 759.699,A -85,B 0,C 180,E1 -31617.752,E2 -31617.752} C_VEL
LIN {X 0,Y 117.722,Z 759.301,A -85,B 0,C 180,E1 -31618.56,E2 -31618.56} C_VEL
LIN {X 0,Y 109.309,Z 753.644,A -85,B 0,C 180,E1 -31629.511,E2 -31629.511} C_VEL
LIN {X 0,Y 106.105,Z 748.351,A -85,B 0,C 180,E1 -31638.522,E2 -31638.522} C_VEL
LIN {X 0,Y 105.697,Z 741.928,A -85,B 0,C 180,E1 -31647.866,E2 -31647.866} C_VEL
LIN {X 0,Y 107.747,Z 735.158,A -85,B 0,C 180,E1 -31655.946,E2 -31655.946} C_VEL
LIN {X 0,Y 109.739,Z 731.068,A -85,B 0,C 180,E1 -31660.156,E2 -31660.156} C_VEL
LIN {X 0,Y 108.049,Z 732.272,A -85,B 0,C 180,E1 -31660.583,E2 -31660.583} C_VEL
LIN {X 0,Y 99.206,Z 739.898,A -85,B 0,C 180,E1 -31659.597,E2 -31659.597} C_VEL
LIN {X 0,Y 90.772,Z 746.261,A -85,B 0,C 180,E1 -31658.291,E2 -31658.291} C_VEL
LIN {X 0,Y 80.548,Z 752.795,A -85,B 0,C 180,E1 -31656.367,E2 -31656.367} C_VEL
LIN {X 0,Y 70.38,Z 758.227,A -85,B 0,C 180,E1 -31653.987,E2 -31653.987} C_VEL
LIN {X 0,Y 60.358,Z 762.676,A -85,B 0,C 180,E1 -31650.841,E2 -31650.841} C_VEL
LIN {X 0,Y 50.579,Z 766.229,A -85,B 0,C 180,E1 -31646.48,E2 -31646.48} C_VEL
LIN {X 0,Y 44.279,Z 768.178,A -85,B 0,C 180,E1 -31642.522,E2 -31642.522} C_VEL
LIN {X 0,Y 32.802,Z 770.883,A -85,B 0,C 180,E1 -31629.997,E2 -31629.997} C_VEL
LIN {X 0,Y 24.405,Z 772.207,A -85,B 0,C 180,E1 -31606.737,E2 -31606.737} C_VEL
LIN {X 0,Y 22.718,Z 772.475,A -85,B 0,C 180,E1 -31590,E2 -31590} C_VEL
LIN {X 0,Y 28.005,Z 771.716,A -85,B 0,C 180,E1 -31559.874,E2 -31559.874} C_VEL
LIN {X 0,Y 32.805,Z 770.883,A -85,B 0,C 180,E1 -31550.007,E2 -31550.007} C_VEL
LIN {X 0,Y 44.304,Z 768.177,A -85,B 0,C 180,E1 -31537.521,E2 -31537.521} C_VEL
LIN {X 0,Y 53.508,Z 765.326,A -85,B 0,C 180,E1 -31532.097,E2 -31532.097} C_VEL
LIN {X 0,Y 63.674,Z 761.377,A -85,B 0,C 180,E1 -31527.996,E2 -31527.996} C_VEL
LIN {X 0,Y 73.763,Z 756.611,A -85,B 0,C 180,E1 -31525.16,E2 -31525.16} C_VEL
LIN {X 0,Y 85.643,Z 749.671,A -85,B 0,C 180,E1 -31522.605,E2 -31522.605} C_VEL
LIN {X 0,Y 94.196,Z 743.802,A -85,B 0,C 180,E1 -31521.156,E2 -31521.156} C_VEL
LIN {X 0,Y 103.242,Z 736.562,A -85,B 0,C 180,E1 -31519.897,E2 -31519.897} C_VEL
LIN {X 0,Y 108.017,Z 732.275,A -85,B 0,C 180,E1 -31519.369,E2 -31519.369} C_VEL
LIN {X 0,Y 109.809,Z 730.975,A -85,B 0,C 180,E1 -31519.78,E2 -31519.78} C_VEL
LIN {X 0,Y 106.267,Z 739.442,A -85,B 0,C 180,E1 -31528.978,E2 -31528.978} C_VEL
LIN {X 0,Y 105.542,Z 745.428,A -85,B 0,C 180,E1 -31536.96,E2 -31536.96} C_VEL
LIN {X 0,Y 107.364,Z 751.156,A -85,B 0,C 180,E1 -31546.056,E2 -31546.056} C_VEL
LIN {X 0,Y 112.751,Z 756.495,A -85,B 0,C 180,E1 -31555.877,E2 -31555.877} C_VEL
LIN {X 0,Y 118.853,Z 759.782,A -85,B 0,C 180,E1 -31562.492,E2 -31562.492} C_VEL
LIN {X 0,Y 131.242,Z 763.558,A -85,B 0,C 180,E1 -31571.259,E2 -31571.259} C_VEL
LIN {X 0,Y 144.054,Z 765.814,A -85,B 0,C 180,E1 -31577.347,E2 -31577.347} C_VEL
LIN {X 0,Y 157.745,Z 767.24,A -85,B 0,C 180,E1 -31582.319,E2 -31582.319} C_VEL
LIN {X 0,Y 169.117,Z 767.885,A -85,B 0,C 180,E1 -31585.822,E2 -31585.822} C_VEL
LIN {X 0,Y 175.826,Z 768.012,A -85,B 0,C 180,E1 -31587.798,E2 -31587.798} C_VEL
LIN {X 0,Y 182.456,Z 768.019,A -85,B 0,C 180,E1 -31590,E2 -31590} C_VEL
LIN {X 0,Y 175.52,Z 768.011,A -85,B 0,C 180,E1 -31592.295,E2 -31592.295} C_VEL
LIN {X 0,Y 166.97,Z 767.786,A -85,B 0,C 180,E1 -31594.829,E2 -31594.829} C_VEL
LIN {X 0,Y 150.026,Z 766.508,A -85,B 0,C 180,E1 -31600.352,E2 -31600.352} C_VEL
LIN {X 0,Y 134.527,Z 764.215,A -85,B 0,C 180,E1 -31606.995,E2 -31606.995} C_VEL
LIN {X 0,Y 123.096,Z 761.316,A -85,B 0,C 180,E1 -31614.011,E2 -31614.011} C_VEL
LIN {X 0,Y 117.722,Z 759.301,A -85,B 0,C 180,E1 -31618.56,E2 -31618.56} C_VEL
LIN {X 0,Y 114.661,Z 758.249,A -85,B 0,C 180,E1 -31621.001,E2 -31621.001} C_VEL
LIN {X 0,Y 104.159,Z 756.174,A -85,B 0,C 180,E1 -31628.496,E2 -31628.496} C_VEL
LIN {X 0,Y 101.789,Z 755.048,A -85,B 0,C 180,E1 -31631.431,E2 -31631.431} C_VEL
LIN {X 0,Y 101.302,Z 754.521,A -85,B 0,C 180,E1 -31632.466,E2 -31632.466} C_VEL
LIN {X 0,Y 99.281,Z 749.229,A -85,B 0,C 180,E1 -31642.292,E2 -31642.292} C_VEL
LIN {X 0,Y 99.972,Z 743.996,A -85,B 0,C 180,E1 -31650.524,E2 -31650.524} C_VEL
LIN {X 0,Y 101.407,Z 740.26,A -85,B 0,C 180,E1 -31655.431,E2 -31655.431} C_VEL
LIN {X 0,Y 100.351,Z 740.932,A -85,B 0,C 180,E1 -31655.564,E2 -31655.564} C_VEL
LIN {X 0,Y 91.961,Z 747.199,A -85,B 0,C 180,E1 -31653.891,E2 -31653.891} C_VEL
LIN {X 0,Y 83.662,Z 752.596,A -85,B 0,C 180,E1 -31651.889,E2 -31651.889} C_VEL
LIN {X 0,Y 73.793,Z 758.028,A -85,B 0,C 180,E1 -31648.997,E2 -31648.997} C_VEL
LIN {X 0,Y 64.14,Z 762.477,A -85,B 0,C 180,E1 -31645.263,E2 -31645.263} C_VEL
LIN {X 0,Y 54.844,Z 766.03,A -85,B 0,C 180,E1 -31640.252,E2 -31640.252} C_VEL
LIN {X 0,Y 48.955,Z 767.979,A -85,B 0,C 180,E1 -31635.872,E2 -31635.872} C_VEL
LIN {X 0,Y 38.539,Z 770.685,A -85,B 0,C 180,E1 -31623.167,E2 -31623.167} C_VEL
LIN {X 0,Y 31.294,Z 772.008,A -85,B 0,C 180,E1 -31602.978,E2 -31602.978} C_VEL
LIN {X 0,Y 29.83,Z 772.276,A -85,B 0,C 180,E1 -31590,E2 -31590} C_VEL
LIN {X 0,Y 34.384,Z 771.516,A -85,B 0,C 180,E1 -31565.871,E2 -31565.871} C_VEL
LIN {X 0,Y 38.544,Z 770.684,A -85,B 0,C 180,E1 -31556.839,E2 -31556.839} C_VEL
LIN {X 0,Y 48.99,Z 767.978,A -85,B 0,C 180,E1 -31544.17,E2 -31544.17} C_VEL
LIN {X 0,Y 61.02,Z 763.745,A -85,B 0,C 180,E1 -31536.272,E2 -31536.272} C_VEL
LIN {X 0,Y 70.559,Z 759.608,A -85,B 0,C 180,E1 -31532.154,E2 -31532.154} C_VEL
LIN {X 0,Y 80.38,Z 754.507,A -85,B 0,C 180,E1 -31529.035,E2 -31529.035} C_VEL
LIN {X 0,Y 90.276,Z 748.337,A -85,B 0,C 180,E1 -31526.459,E2 -31526.459} C_VEL
LIN {X 0,Y 98.651,Z 742.269,A -85,B 0,C 180,E1 -31524.728,E2 -31524.728} C_VEL
LIN {X 0,Y 100.334,Z 740.933,A -85,B 0,C 180,E1 -31524.415,E2 -31524.415} C_VEL
LIN {X 0,Y 101.408,Z 740.259,A -85,B 0,C 180,E1 -31524.569,E2 -31524.569} C_VEL
LIN {X 0,Y 99.501,Z 745.725,A -85,B 0,C 180,E1 -31532.052,E2 -31532.052} C_VEL
LIN {X 0,Y 99.75,Z 751.66,A -85,B 0,C 180,E1 -31542.013,E2 -31542.013} C_VEL
LIN {X 0,Y 103.465,Z 756.809,A -85,B 0,C 180,E1 -31552.315,E2 -31552.315} C_VEL
LIN {X 0,Y 107.644,Z 759.651,A -85,B 0,C 180,E1 -31558.513,E2 -31558.513} C_VEL
LIN {X 0,Y 115.285,Z 762.73,A -85,B 0,C 180,E1 -31566.121,E2 -31566.121} C_VEL
LIN {X 0,Y 130.597,Z 766.022,A -85,B 0,C 180,E1 -31575.61,E2 -31575.61} C_VEL
LIN {X 0,Y 148.737,Z 767.794,A -85,B 0,C 180,E1 -31582.86,E2 -31582.86} C_VEL
LIN {X 0,Y 164.072,Z 768.325,A -85,B 0,C 180,E1 -31587.545,E2 -31587.545} C_VEL
LIN {X 0,Y 172.44,Z 768.299,A -85,B 0,C 180,E1 -31590,E2 -31590} C_VEL
LIN {X 0,Y 164.112,Z 768.324,A -85,B 0,C 180,E1 -31592.454,E2 -31592.454} C_VEL
LIN {X 0,Y 148.741,Z 767.791,A -85,B 0,C 180,E1 -31597.152,E2 -31597.152} C_VEL
LIN {X 0,Y 130.598,Z 766.021,A -85,B 0,C 180,E1 -31604.391,E2 -31604.391} C_VEL
LIN {X 0,Y 115.288,Z 762.727,A -85,B 0,C 180,E1 -31613.883,E2 -31613.883} C_VEL
LIN {X 0,Y 105.824,Z 758.537,A -85,B 0,C 180,E1 -31623.889,E2 -31623.889} C_VEL
LIN {X 0,Y 101.302,Z 754.521,A -85,B 0,C 180,E1 -31632.466,E2 -31632.466} C_VEL
LIN {X 0,Y 99.967,Z 753.69,A -85,B 0,C 180,E1 -31634.555,E2 -31634.555} C_VEL
LIN {X 0,Y 93.492,Z 752.403,A -85,B 0,C 180,E1 -31641.536,E2 -31641.536} C_VEL
LIN {X 0,Y 92.835,Z 751.497,A -85,B 0,C 180,E1 -31643.879,E2 -31643.879} C_VEL
LIN {X 0,Y 93.286,Z 748.683,A -85,B 0,C 180,E1 -31648.977,E2 -31648.977} C_VEL
LIN {X 0,Y 90.453,Z 750.41,A -85,B 0,C 180,E1 -31648.721,E2 -31648.721} C_VEL
LIN {X 0,Y 80.88,Z 756.213,A -85,B 0,C 180,E1 -31645.636,E2 -31645.636} C_VEL
LIN {X 0,Y 71.519,Z 760.978,A -85,B 0,C 180,E1 -31641.825,E2 -31641.825} C_VEL
LIN {X 0,Y 59.66,Z 765.831,A -85,B 0,C 180,E1 -31634.974,E2 -31634.974} C_VEL
LIN {X 0,Y 54.185,Z 767.779,A -85,B 0,C 180,E1 -31630.429,E2 -31630.429} C_VEL
LIN {X 0,Y 44.677,Z 770.486,A -85,B 0,C 180,E1 -31618.158,E2 -31618.158} C_VEL
LIN {X 0,Y 38.298,Z 771.808,A -85,B 0,C 180,E1 -31600.574,E2 -31600.574} C_VEL
LIN {X 0,Y 36.932,Z 772.078,A -85,B 0,C 180,E1 -31590,E2 -31590} C_VEL
LIN {X 0,Y 41.018,Z 771.317,A -85,B 0,C 180,E1 -31569.96,E2 -31569.96} C_VEL
LIN {X 0,Y 44.686,Z 770.485,A -85,B 0,C 180,E1 -31561.848,E2 -31561.848} C_VEL
LIN {X 0,Y 54.231,Z 767.778,A -85,B 0,C 180,E1 -31549.613,E2 -31549.613} C_VEL
LIN {X 0,Y 65.501,Z 763.546,A -85,B 0,C 180,E1 -31541.318,E2 -31541.318} C_VEL
LIN {X 0,Y 74.602,Z 759.408,A -85,B 0,C 180,E1 -31536.799,E2 -31536.799} C_VEL
LIN {X 0,Y 84.076,Z 754.308,A -85,B 0,C 180,E1 -31533.292,E2 -31533.292} C_VEL
LIN {X 0,Y 90.452,Z 750.41,A -85,B 0,C 180,E1 -31531.277,E2 -31531.277} C_VEL
LIN {X 0,Y 93.284,Z 748.684,A -85,B 0,C 180,E1 -31531.023,E2 -31531.023} C_VEL
LIN {X 0,Y 93.339,Z 754.715,A -85,B 0,C 180,E1 -31542.658,E2 -31542.658} C_VEL
LIN {X 0,Y 98.003,Z 759.972,A -85,B 0,C 180,E1 -31554.993,E2 -31554.993} C_VEL
LIN {X 0,Y 108.404,Z 764.231,A -85,B 0,C 180,E1 -31567.109,E2 -31567.109} C_VEL
LIN {X 0,Y 117.329,Z 766.186,A -85,B 0,C 180,E1 -31573.409,E2 -31573.409} C_VEL
LIN {X 0,Y 134.932,Z 768.075,A -85,B 0,C 180,E1 -31581.729,E2 -31581.729} C_VEL
LIN {X 0,Y 151.949,Z 768.659,A -85,B 0,C 180,E1 -31587.349,E2 -31587.349} C_VEL
LIN {X 0,Y 161.4,Z 768.607,A -85,B 0,C 180,E1 -31590,E2 -31590} C_VEL
LIN {X 0,Y 147.922,Z 768.649,A -85,B 0,C 180,E1 -31593.871,E2 -31593.871} C_VEL
LIN {X 0,Y 128.775,Z 767.62,A -85,B 0,C 180,E1 -31600.786,E2 -31600.786} C_VEL
LIN {X 0,Y 115.574,Z 765.868,A -85,B 0,C 180,E1 -31607.7,E2 -31607.7} C_VEL
LIN {X 0,Y 103.304,Z 762.561,A -85,B 0,C 180,E1 -31617.825,E2 -31617.825} C_VEL
LIN {X 0,Y 96.859,Z 759.115,A -85,B 0,C 180,E1 -31627.05,E2 -31627.05} C_VEL
LIN {X 0,Y 93.356,Z 754.703,A -85,B 0,C 180,E1 -31637.352,E2 -31637.352} C_VEL
LIN {X 0,Y 92.835,Z 751.497,A -85,B 0,C 180,E1 -31643.879,E2 -31643.879} C_VEL
LIN {X 0,Y 91.781,Z 752.245,A -85,B 0,C 180,E1 -31643.374,E2 -31643.374} C_VEL
LIN {X 0,Y 90.047,Z 754.515,A -85,B 0,C 180,E1 -31640.392,E2 -31640.392} C_VEL
LIN {X 0,Y 88.92,Z 758.75,A -85,B 0,C 180,E1 -31632.37,E2 -31632.37} C_VEL
LIN {X 0,Y 89.966,Z 760.995,A -85,B 0,C 180,E1 -31626.993,E2 -31626.993} C_VEL
LIN {X 0,Y 90.738,Z 761.552,A -85,B 0,C 180,E1 -31625.251,E2 -31625.251} C_VEL
LIN {X 0,Y 97.655,Z 764.556,A -85,B 0,C 180,E1 -31615.582,E2 -31615.582} C_VEL
LIN {X 0,Y 104.365,Z 766.278,A -85,B 0,C 180,E1 -31609.484,E2 -31609.484} C_VEL
LIN {X 0,Y 121.191,Z 768.355,A -85,B 0,C 180,E1 -31599.661,E2 -31599.661} C_VEL
LIN {X 0,Y 140.694,Z 768.998,A -85,B 0,C 180,E1 -31592.533,E2 -31592.533} C_VEL
LIN {X 0,Y 149.46,Z 768.94,A -85,B 0,C 180,E1 -31590,E2 -31590} C_VEL
LIN {X 0,Y 129.636,Z 768.818,A -85,B 0,C 180,E1 -31583.776,E2 -31583.776} C_VEL
LIN {X 0,Y 115.207,Z 767.834,A -85,B 0,C 180,E1 -31577.426,E2 -31577.426} C_VEL
LIN {X 0,Y 104.021,Z 766.206,A -85,B 0,C 180,E1 -31570.257,E2 -31570.257} C_VEL
LIN {X 0,Y 95.538,Z 763.902,A -85,B 0,C 180,E1 -31561.971,E2 -31561.971} C_VEL
LIN {X 0,Y 88.947,Z 760.288,A -85,B 0,C 180,E1 -31550.795,E2 -31550.795} C_VEL
LIN {X 0,Y 86.367,Z 755.754,A -85,B 0,C 180,E1 -31538.934,E2 -31538.934} C_VEL
LIN {X 0,Y 82.092,Z 757.629,A -85,B 0,C 180,E1 -31539.603,E2 -31539.603} C_VEL
LIN {X 0,Y 73.249,Z 762.078,A -85,B 0,C 180,E1 -31543.98,E2 -31543.98} C_VEL
LIN {X 0,Y 64.985,Z 765.629,A -85,B 0,C 180,E1 -31549.543,E2 -31549.543} C_VEL
LIN {X 0,Y 59.871,Z 767.578,A -85,B 0,C 180,E1 -31554.062,E2 -31554.062} C_VEL
LIN {X 0,Y 51.111,Z 770.286,A -85,B 0,C 180,E1 -31565.638,E2 -31565.638} C_VEL
LIN {X 0,Y 45.347,Z 771.609,A -85,B 0,C 180,E1 -31581.084,E2 -31581.084} C_VEL
LIN {X 0,Y 44.062,Z 771.879,A -85,B 0,C 180,E1 -31590,E2 -31590} C_VEL
LIN {X 0,Y 47.797,Z 771.117,A -85,B 0,C 180,E1 -31607.102,E2 -31607.102} C_VEL
LIN {X 0,Y 51.099,Z 770.286,A -85,B 0,C 180,E1 -31614.368,E2 -31614.368} C_VEL
LIN {X 0,Y 59.812,Z 767.58,A -85,B 0,C 180,E1 -31625.979,E2 -31625.979} C_VEL
LIN {X 0,Y 70.392,Z 763.347,A -85,B 0,C 180,E1 -31634.336,E2 -31634.336} C_VEL
LIN {X 0,Y 79.095,Z 759.209,A -85,B 0,C 180,E1 -31639.048,E2 -31639.048} C_VEL
LIN {X 0,Y 82.092,Z 757.629,A -85,B 0,C 180,E1 -31640.397,E2 -31640.397} C_VEL
LIN {X 0,Y 86.382,Z 755.744,A -85,B 0,C 180,E1 -31641.074,E2 -31641.074} C_VEL
LIN {X 0,Y 89.373,Z 760.641,A -85,B 0,C 180,E1 -31628.156,E2 -31628.156} C_VEL
LIN {X 0,Y 90.738,Z 761.552,A -85,B 0,C 180,E1 -31625.251,E2 -31625.251} C_VEL
LIN {X 0,Y 92.099,Z 762.866,A -85,B 0,C 180,E1 -31621.725,E2 -31621.725} C_VEL
LIN {X 0,Y 93.486,Z 765.066,A -85,B 0,C 180,E1 -31615.806,E2 -31615.806} C_VEL
LIN {X 0,Y 95.923,Z 766.921,A -85,B 0,C 180,E1 -31610.12,E2 -31610.12} C_VEL
LIN {X 0,Y 98.799,Z 767.553,A -85,B 0,C 180,E1 -31607.131,E2 -31607.131} C_VEL
LIN {X 0,Y 113.667,Z 768.975,A -85,B 0,C 180,E1 -31598.411,E2 -31598.411} C_VEL
LIN {X 0,Y 126.872,Z 769.348,A -85,B 0,C 180,E1 -31593.175,E2 -31593.175} C_VEL
LIN {X 0,Y 137.079,Z 769.285,A -85,B 0,C 180,E1 -31590,E2 -31590} C_VEL
LIN {X 0,Y 117.014,Z 769.168,A -85,B 0,C 180,E1 -31583.101,E2 -31583.101} C_VEL
LIN {X 0,Y 101.832,Z 767.993,A -85,B 0,C 180,E1 -31575.057,E2 -31575.057} C_VEL
LIN {X 0,Y 91.834,Z 766.25,A -85,B 0,C 180,E1 -31566.681,E2 -31566.681} C_VEL
LIN {X 0,Y 83.13,Z 762.883,A -85,B 0,C 180,E1 -31553.717,E2 -31553.717} C_VEL
LIN {X 0,Y 80.818,Z 760.999,A -85,B 0,C 180,E1 -31547.033,E2 -31547.033} C_VEL
LIN {X 0,Y 77.589,Z 762.253,A -85,B 0,C 180,E1 -31548.243,E2 -31548.243} C_VEL
LIN {X 0,Y 70.586,Z 765.43,A -85,B 0,C 180,E1 -31553.317,E2 -31553.317} C_VEL
LIN {X 0,Y 65.821,Z 767.377,A -85,B 0,C 180,E1 -31557.733,E2 -31557.733} C_VEL
LIN {X 0,Y 57.703,Z 770.086,A -85,B 0,C 180,E1 -31568.569,E2 -31568.569} C_VEL
LIN {X 0,Y 52.413,Z 771.41,A -85,B 0,C 180,E1 -31582.294,E2 -31582.294} C_VEL
LIN {X 0,Y 51.183,Z 771.681,A -85,B 0,C 180,E1 -31590,E2 -31590} C_VEL
LIN {X 0,Y 54.673,Z 770.918,A -85,B 0,C 180,E1 -31604.897,E2 -31604.897} C_VEL
LIN {X 0,Y 57.689,Z 770.087,A -85,B 0,C 180,E1 -31611.436,E2 -31611.436} C_VEL
LIN {X 0,Y 65.735,Z 767.38,A -85,B 0,C 180,E1 -31622.314,E2 -31622.314} C_VEL
LIN {X 0,Y 73.039,Z 764.413,A -85,B 0,C 180,E1 -31628.714,E2 -31628.714} C_VEL
LIN {X 0,Y 78.947,Z 761.621,A -85,B 0,C 180,E1 -31632.585,E2 -31632.585} C_VEL
LIN {X 0,Y 80.879,Z 761.008,A -85,B 0,C 180,E1 -31632.892,E2 -31632.892} C_VEL
LIN {X 0,Y 87.744,Z 765.034,A -85,B 0,C 180,E1 -31618.234,E2 -31618.234} C_VEL
LIN {X 0,Y 96.564,Z 767.218,A -85,B 0,C 180,E1 -31608.895,E2 -31608.895} C_VEL
LIN {X 0,Y 98.799,Z 767.553,A -85,B 0,C 180,E1 -31607.131,E2 -31607.131} C_VEL
LIN {X 0,Y 101.974,Z 768.205,A -85,B 0,C 180,E1 -31604.303,E2 -31604.303} C_VEL
LIN {X 0,Y 110.374,Z 769.62,A -85,B 0,C 180,E1 -31595.831,E2 -31595.831} C_VEL
LIN {X 0,Y 114.249,Z 769.698,A -85,B 0,C 180,E1 -31593.567,E2 -31593.567} C_VEL
LIN {X 0,Y 115.762,Z 769.693,A -85,B 0,C 180,E1 -31592.943,E2 -31592.943} C_VEL
LIN {X 0,Y 124.405,Z 769.639,A -85,B 0,C 180,E1 -31590,E2 -31590} C_VEL
LIN {X 0,Y 104.592,Z 769.512,A -85,B 0,C 180,E1 -31582.277,E2 -31582.277} C_VEL
LIN {X 0,Y 94.131,Z 768.842,A -85,B 0,C 180,E1 -31576.063,E2 -31576.063} C_VEL
LIN {X 0,Y 82.217,Z 766.857,A -85,B 0,C 180,E1 -31564.698,E2 -31564.698} C_VEL
LIN {X 0,Y 77.419,Z 765.198,A -85,B 0,C 180,E1 -31556.999,E2 -31556.999} C_VEL
LIN {X 0,Y 76.449,Z 765.23,A -85,B 0,C 180,E1 -31556.525,E2 -31556.525} C_VEL
LIN {X 0,Y 71.987,Z 767.177,A -85,B 0,C 180,E1 -31560.782,E2 -31560.782} C_VEL
LIN {X 0,Y 64.411,Z 769.887,A -85,B 0,C 180,E1 -31570.893,E2 -31570.893} C_VEL
LIN {X 0,Y 59.489,Z 771.211,A -85,B 0,C 180,E1 -31583.215,E2 -31583.215} C_VEL
LIN {X 0,Y 58.296,Z 771.482,A -85,B 0,C 180,E1 -31590,E2 -31590} C_VEL
LIN {X 0,Y 61.612,Z 770.719,A -85,B 0,C 180,E1 -31603.187,E2 -31603.187} C_VEL
LIN {X 0,Y 64.394,Z 769.887,A -85,B 0,C 180,E1 -31609.112,E2 -31609.112} C_VEL
LIN {X 0,Y 71.898,Z 767.18,A -85,B 0,C 180,E1 -31619.258,E2 -31619.258} C_VEL
LIN {X 0,Y 76.36,Z 765.233,A -85,B 0,C 180,E1 -31623.519,E2 -31623.519} C_VEL
LIN {X 0,Y 77.418,Z 765.198,A -85,B 0,C 180,E1 -31623.002,E2 -31623.002} C_VEL
LIN {X 0,Y 84.019,Z 767.287,A -85,B 0,C 180,E1 -31613.062,E2 -31613.062} C_VEL
LIN {X 0,Y 95.976,Z 768.981,A -85,B 0,C 180,E1 -31602.69,E2 -31602.69} C_VEL
LIN {X 0,Y 112.732,Z 769.7,A -85,B 0,C 180,E1 -31594.096,E2 -31594.096} C_VEL
LIN {X 0,Y 115.762,Z 769.693,A -85,B 0,C 180,E1 -31592.943,E2 -31592.943} C_VEL
LIN {X 0,Y 116.258,Z 769.727,A -85,B 0,C 180,E1 -31592.347,E2 -31592.347} C_VEL
LIN {X 0,Y 115.507,Z 769.832,A -85,B 0,C 180,E1 -31591.19,E2 -31591.19} C_VEL
LIN {X 0,Y 112.562,Z 769.958,A -85,B 0,C 180,E1 -31589.616,E2 -31589.616} C_VEL
LIN {X 0,Y 100.024,Z 770.045,A -85,B 0,C 180,E1 -31585.299,E2 -31585.299} C_VEL
LIN {X 0,Y 84.27,Z 769.312,A -85,B 0,C 180,E1 -31575.511,E2 -31575.511} C_VEL
LIN {X 0,Y 76.21,Z 768.143,A -85,B 0,C 180,E1 -31567.242,E2 -31567.242} C_VEL
LIN {X 0,Y 74.491,Z 768.443,A -85,B 0,C 180,E1 -31567.828,E2 -31567.828} C_VEL
LIN {X 0,Y 71.2,Z 769.688,A -85,B 0,C 180,E1 -31572.776,E2 -31572.776} C_VEL
LIN {X 0,Y 66.592,Z 771.012,A -85,B 0,C 180,E1 -31583.942,E2 -31583.942} C_VEL
LIN {X 0,Y 65.433,Z 771.283,A -85,B 0,C 180,E1 -31590,E2 -31590} C_VEL
LIN {X 0,Y 68.591,Z 770.519,A -85,B 0,C 180,E1 -31601.825,E2 -31601.825} C_VEL
LIN {X 0,Y 71.18,Z 769.688,A -85,B 0,C 180,E1 -31607.229,E2 -31607.229} C_VEL
LIN {X 0,Y 74.441,Z 768.445,A -85,B 0,C 180,E1 -31612.187,E2 -31612.187} C_VEL
LIN {X 0,Y 76.207,Z 768.144,A -85,B 0,C 180,E1 -31612.753,E2 -31612.753} C_VEL
LIN {X 0,Y 86.465,Z 769.466,A -85,B 0,C 180,E1 -31602.751,E2 -31602.751} C_VEL
LIN {X 0,Y 101.679,Z 770.041,A -85,B 0,C 180,E1 -31593.963,E2 -31593.963} C_VEL
LIN {X 0,Y 111.726,Z 769.992,A -85,B 0,C 180,E1 -31590,E2 -31590} C_VEL
LIN {X 0,Y 100.024,Z 770.045,A -85,B 0,C 180,E1 -31585.299,E2 -31585.299} C_VEL
LIN {X 0,Y 96.573,Z 770.089,A -85,B 0,C 180,E1 -31584.124,E2 -31584.124} C_VEL
LIN {X 0,Y 83.691,Z 770.289,A -85,B 0,C 180,E1 -31581.536,E2 -31581.536} C_VEL
LIN {X 0,Y 80.456,Z 770.182,A -85,B 0,C 180,E1 -31579.924,E2 -31579.924} C_VEL
LIN {X 0,Y 77.596,Z 769.984,A -85,B 0,C 180,E1 -31577.63,E2 -31577.63} C_VEL
LIN {X 0,Y 75.603,Z 770.32,A -85,B 0,C 180,E1 -31579.286,E2 -31579.286} C_VEL
LIN {X 0,Y 72.559,Z 771.085,A -85,B 0,C 180,E1 -31590,E2 -31590} C_VEL
LIN {X 0,Y 75.595,Z 770.32,A -85,B 0,C 180,E1 -31600.716,E2 -31600.716} C_VEL
LIN {X 0,Y 77.592,Z 769.984,A -85,B 0,C 180,E1 -31602.373,E2 -31602.373} C_VEL
LIN {X 0,Y 91.52,Z 770.38,A -85,B 0,C 180,E1 -31593.384,E2 -31593.384} C_VEL
LIN {X 0,Y 99.097,Z 770.344,A -85,B 0,C 180,E1 -31590,E2 -31590} C_VEL
LIN {X 0,Y 80.456,Z 770.182,A -85,B 0,C 180,E1 -31579.924,E2 -31579.924} C_VEL
LIN {X 0,Y 79.237,Z 770.253,A -85,B 0,C 180,E1 -31579.969,E2 -31579.969} C_VEL
LIN {X 0,Y 77.586,Z 770.532,A -85,B 0,C 180,E1 -31581.524,E2 -31581.524} C_VEL
LIN {X 0,Y 76.579,Z 770.758,A -85,B 0,C 180,E1 -31585.033,E2 -31585.033} C_VEL
LIN {X 0,Y 76.829,Z 770.922,A -85,B 0,C 180,E1 -31588.742,E2 -31588.742} C_VEL
LIN {X 0,Y 78.313,Z 770.863,A -85,B 0,C 180,E1 -31591.948,E2 -31591.948} C_VEL
LIN {X 0,Y 80.09,Z 770.746,A -85,B 0,C 180,E1 -31592.984,E2 -31592.984} C_VEL
LIN {X 0,Y 81.041,Z 770.716,A -85,B 0,C 180,E1 -31592.91,E2 -31592.91} C_VEL
LIN {X 0,Y 86.683,Z 770.691,A -85,B 0,C 180,E1 -31590,E2 -31590} C_VEL
LIN {X 0,Y 81.043,Z 770.717,A -85,B 0,C 180,E1 -31587.11,E2 -31587.11} C_VEL
LIN {X 0,Y 79.891,Z 770.838,A -85,B 0,C 180,E1 -31588.803,E2 -31588.803} C_VEL
LIN {X 0,Y 79.885,Z 770.838,A -85,B 0,C 180,E1 -31591.207,E2 -31591.207} C_VEL
LIN {X 0,Y 81.041,Z 770.716,A -85,B 0,C 180,E1 -31592.91,E2 -31592.91} C_VEL
LIN {X 0,Y 81.041,Z 770.716,A -85,B 0,C 180,E1 -31592.91,E2 -31592.91}

QRS_NEXT_CUT()

QRS_NEXT()
QRS_HOME()

END
